Yaskawa INFORM job: DEMO_ROOF_UPPER_0625_3PAINT_3.JBI

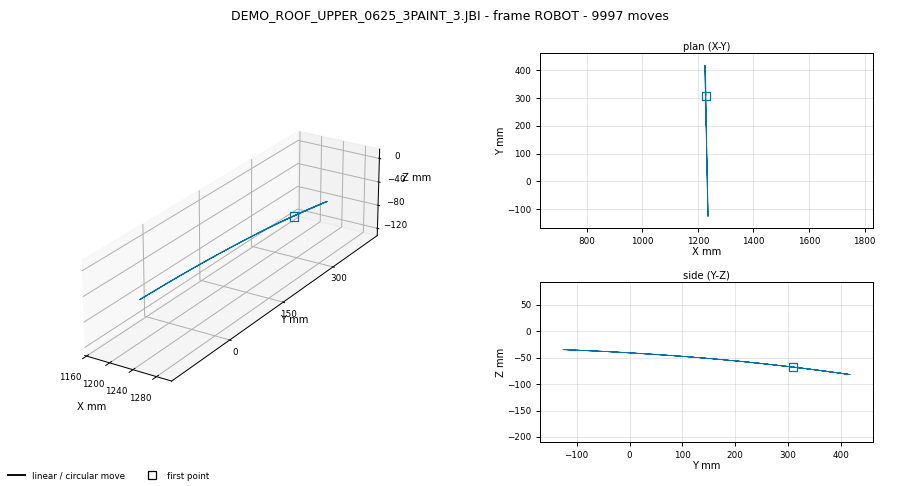
[picture p0: tool path of DEMO_ROOF_UPPER_0625_3PAINT_3.JBI in frame ROBOT, 9997 of 9997 moves have a stored position in this frame; points joined in program order, loops and branches not executed]
/JOB
//NAME DEMO_ROOF_UPPER_0625_3PAINT3
//POS
///NPOS 9997,0,0,0,0,0
///TOOL 0
///USER 0
///POSTYPE ROBOT
///RECTAN
///RCONF 1,0,0,0,0,0,0,0,0,0,0,0,0,0,0,0,0,0,0,0,0,0,0,0
C00000=1229.073,308.460,-67.633,-176.288,6.838,148.176
C00001=1229.069,308.709,-67.663,-176.286,6.841,148.176
C00002=1229.065,308.957,-67.692,-176.284,6.843,148.176
C00003=1229.061,309.205,-67.722,-176.281,6.846,148.176
C00004=1229.056,309.453,-67.752,-176.279,6.848,148.176
C00005=1229.052,309.701,-67.782,-176.277,6.850,148.176
C00006=1229.048,309.950,-67.811,-176.275,6.853,148.176
C00007=1229.044,310.198,-67.841,-176.272,6.856,148.176
C00008=1229.039,310.446,-67.871,-176.270,6.858,148.176
C00009=1229.035,310.694,-67.901,-176.268,6.860,148.176
C00010=1229.031,310.942,-67.930,-176.265,6.863,148.176
C00011=1229.026,311.190,-67.961,-176.263,6.865,148.176
C00012=1229.023,311.439,-67.991,-176.261,6.868,148.176
C00013=1229.019,311.687,-68.021,-176.258,6.871,148.176
C00014=1229.014,311.936,-68.051,-176.256,6.873,148.176
C00015=1229.010,312.184,-68.081,-176.254,6.875,148.176
C00016=1229.006,312.432,-68.111,-176.252,6.877,148.176
C00017=1229.001,312.680,-68.141,-176.249,6.880,148.176
C00018=1228.997,312.928,-68.171,-176.247,6.883,148.176
C00019=1228.992,313.176,-68.201,-176.245,6.885,148.176
C00020=1228.988,313.424,-68.231,-176.243,6.888,148.176
C00021=1228.984,313.672,-68.261,-176.241,6.890,148.176
C00022=1228.979,313.920,-68.291,-176.239,6.893,148.176
C00023=1228.975,314.168,-68.321,-176.237,6.895,148.176
C00024=1228.971,314.416,-68.352,-176.234,6.898,148.176
C00025=1228.966,314.665,-68.381,-176.232,6.900,148.176
C00026=1228.963,314.912,-68.411,-176.230,6.902,148.176
C00027=1228.957,315.189,-68.445,-176.227,6.905,148.176
C00028=1228.953,315.465,-68.478,-176.224,6.909,148.176
C00029=1228.948,315.741,-68.512,-176.222,6.911,148.176
C00030=1228.944,316.015,-68.545,-176.220,6.914,148.176
C00031=1228.939,316.264,-68.575,-176.218,6.916,148.176
C00032=1228.935,316.512,-68.606,-176.215,6.919,148.176
C00033=1228.931,316.761,-68.636,-176.213,6.922,148.176
C00034=1228.927,317.009,-68.666,-176.211,6.924,148.176
C00035=1228.922,317.257,-68.697,-176.209,6.927,148.176
C00036=1228.918,317.505,-68.726,-176.206,6.929,148.176
C00037=1228.913,317.753,-68.757,-176.204,6.931,148.176
C00038=1228.909,318.000,-68.787,-176.202,6.935,148.176
C00039=1228.905,318.250,-68.818,-176.200,6.937,148.176
C00040=1228.901,318.497,-68.848,-176.198,6.939,148.176
C00041=1228.897,318.745,-68.879,-176.196,6.941,148.176
C00042=1228.892,318.994,-68.908,-176.193,6.944,148.176
C00043=1228.888,319.242,-68.939,-176.192,6.947,148.176
C00044=1228.883,319.489,-68.970,-176.190,6.949,148.176
C00045=1228.880,319.738,-68.999,-176.187,6.952,148.176
C00046=1228.875,319.986,-69.030,-176.185,6.954,148.176
C00047=1228.871,320.234,-69.060,-176.183,6.957,148.176
C00048=1228.867,320.482,-69.091,-176.180,6.960,148.176
C00049=1228.863,320.730,-69.121,-176.178,6.962,148.176
C00050=1228.858,320.979,-69.152,-176.176,6.965,148.176
C00051=1228.854,321.227,-69.182,-176.174,6.968,148.176
C00052=1228.850,321.475,-69.213,-176.172,6.970,148.176
C00053=1228.845,321.722,-69.243,-176.170,6.972,148.176
C00054=1228.841,321.971,-69.275,-176.168,6.975,148.176
C00055=1228.837,322.219,-69.305,-176.165,6.978,148.176
C00056=1228.832,322.467,-69.335,-176.164,6.980,148.176
C00057=1228.829,322.715,-69.365,-176.161,6.982,148.176
C00058=1228.824,322.963,-69.396,-176.159,6.985,148.176
C00059=1228.820,323.212,-69.427,-176.157,6.988,148.176
C00060=1228.816,323.459,-69.457,-176.155,6.990,148.176
C00061=1228.811,323.707,-69.488,-176.152,6.993,148.176
C00062=1228.807,323.955,-69.519,-176.151,6.996,148.176
C00063=1228.803,324.204,-69.550,-176.149,6.998,148.176
C00064=1228.799,324.452,-69.580,-176.146,7.001,148.176
C00065=1228.794,324.699,-69.611,-176.144,7.003,148.176
C00066=1228.790,324.948,-69.642,-176.142,7.006,148.177
C00067=1228.786,325.196,-69.672,-176.140,7.008,148.177
C00068=1228.782,325.444,-69.703,-176.138,7.011,148.177
C00069=1228.777,325.692,-69.733,-176.136,7.014,148.177
C00070=1228.773,325.940,-69.765,-176.134,7.016,148.177
C00071=1228.769,326.188,-69.795,-176.132,7.019,148.177
C00072=1228.765,326.436,-69.825,-176.130,7.021,148.177
C00073=1228.761,326.685,-69.857,-176.127,7.024,148.177
C00074=1228.756,326.933,-69.887,-176.125,7.027,148.177
C00075=1228.752,327.180,-69.918,-176.123,7.029,148.177
C00076=1228.748,327.429,-69.949,-176.121,7.032,148.177
C00077=1228.744,327.677,-69.979,-176.119,7.035,148.177
C00078=1228.739,327.925,-70.010,-176.117,7.037,148.177
C00079=1228.735,328.173,-70.041,-176.115,7.040,148.177
C00080=1228.731,328.420,-70.072,-176.113,7.042,148.177
C00081=1228.727,328.668,-70.103,-176.111,7.045,148.177
C00082=1228.723,328.917,-70.134,-176.109,7.047,148.177
C00083=1228.718,329.165,-70.165,-176.107,7.050,148.177
C00084=1228.714,329.413,-70.196,-176.105,7.053,148.178
C00085=1228.710,329.662,-70.227,-176.102,7.055,148.178
C00086=1228.706,329.909,-70.258,-176.101,7.058,148.178
C00087=1228.701,330.157,-70.288,-176.098,7.061,148.178
C00088=1228.697,330.405,-70.320,-176.097,7.063,148.178
C00089=1228.693,330.653,-70.350,-176.094,7.066,148.178
C00090=1228.688,330.901,-70.382,-176.093,7.068,148.178
C00091=1228.684,331.149,-70.413,-176.090,7.071,148.178
C00092=1228.680,331.397,-70.444,-176.089,7.074,148.178
C00093=1228.676,331.646,-70.475,-176.086,7.076,148.178
C00094=1228.671,331.893,-70.506,-176.084,7.079,148.178
C00095=1228.667,332.141,-70.537,-176.082,7.082,148.178
C00096=1228.664,332.390,-70.568,-176.081,7.084,148.179
C00097=1228.659,332.637,-70.599,-176.078,7.087,148.179
C00098=1228.655,332.886,-70.630,-176.076,7.090,148.179
C00099=1228.651,333.133,-70.661,-176.074,7.092,148.179
C00100=1228.646,333.381,-70.692,-176.073,7.094,148.179
C00101=1228.642,333.629,-70.724,-176.070,7.098,148.179
C00102=1228.638,333.877,-70.754,-176.068,7.100,148.179
C00103=1228.634,334.125,-70.786,-176.066,7.102,148.179
C00104=1228.629,334.373,-70.817,-176.064,7.106,148.179
C00105=1228.625,334.622,-70.848,-176.062,7.108,148.179
C00106=1228.621,334.869,-70.880,-176.060,7.110,148.179
C00107=1228.616,335.117,-70.910,-176.058,7.114,148.180
C00108=1228.613,335.365,-70.942,-176.056,7.116,148.180
C00109=1228.608,335.613,-70.973,-176.054,7.119,148.180
C00110=1228.604,335.861,-71.005,-176.052,7.121,148.180
C00111=1228.600,336.109,-71.036,-176.050,7.124,148.180
C00112=1228.596,336.357,-71.067,-176.048,7.127,148.180
C00113=1228.591,336.605,-71.098,-176.046,7.129,148.180
C00114=1228.588,336.853,-71.130,-176.044,7.132,148.180
C00115=1228.583,337.101,-71.161,-176.042,7.134,148.180
C00116=1228.579,337.350,-71.193,-176.040,7.137,148.181
C00117=1228.574,337.598,-71.224,-176.039,7.140,148.181
C00118=1228.570,337.846,-71.256,-176.036,7.143,148.181
C00119=1228.566,338.094,-71.287,-176.035,7.145,148.181
C00120=1228.562,338.342,-71.318,-176.033,7.148,148.181
C00121=1228.557,338.590,-71.349,-176.030,7.151,148.181
C00122=1228.554,338.838,-71.381,-176.029,7.153,148.181
C00123=1228.549,339.085,-71.413,-176.027,7.156,148.181
C00124=1228.545,339.334,-71.444,-176.025,7.158,148.181
C00125=1228.541,339.581,-71.475,-176.023,7.161,148.182
C00126=1228.537,339.829,-71.508,-176.021,7.164,148.182
C00127=1228.532,340.077,-71.538,-176.020,7.166,148.182
C00128=1228.528,340.325,-71.570,-176.017,7.169,148.182
C00129=1228.524,340.573,-71.602,-176.015,7.172,148.182
C00130=1228.520,340.821,-71.633,-176.014,7.175,148.182
C00131=1228.516,341.099,-71.668,-176.011,7.178,148.182
C00132=1228.510,341.377,-71.704,-176.009,7.180,148.183
C00133=1228.505,341.654,-71.739,-176.007,7.184,148.183
C00134=1228.501,341.932,-71.775,-176.005,7.187,148.183
C00135=1228.497,342.180,-71.805,-176.003,7.189,148.183
C00136=1228.493,342.428,-71.837,-176.001,7.192,148.183
C00137=1228.488,342.675,-71.869,-175.999,7.195,148.183
C00138=1228.484,342.923,-71.901,-175.998,7.198,148.184
C00139=1228.480,343.171,-71.933,-175.996,7.200,148.184
C00140=1228.476,343.419,-71.964,-175.994,7.202,148.184
C00141=1228.471,343.668,-71.996,-175.992,7.206,148.184
C00142=1228.467,343.915,-72.028,-175.990,7.208,148.184
C00143=1228.463,344.163,-72.060,-175.988,7.211,148.184
C00144=1228.459,344.410,-72.091,-175.987,7.213,148.185
C00145=1228.454,344.659,-72.123,-175.984,7.216,148.185
C00146=1228.451,344.907,-72.155,-175.982,7.219,148.185
C00147=1228.446,345.155,-72.186,-175.981,7.221,148.185
C00148=1228.443,345.403,-72.218,-175.979,7.224,148.185
C00149=1228.437,345.651,-72.250,-175.977,7.227,148.185
C00150=1228.434,345.899,-72.282,-175.975,7.230,148.185
C00151=1228.430,346.147,-72.314,-175.974,7.232,148.186
C00152=1228.425,346.394,-72.346,-175.972,7.235,148.186
C00153=1228.421,346.643,-72.377,-175.970,7.238,148.186
C00154=1228.417,346.891,-72.409,-175.968,7.240,148.186
C00155=1228.412,347.139,-72.441,-175.966,7.243,148.186
C00156=1228.409,347.387,-72.473,-175.965,7.246,148.186
C00157=1228.404,347.634,-72.504,-175.962,7.249,148.187
C00158=1228.400,347.882,-72.537,-175.961,7.251,148.187
C00159=1228.396,348.130,-72.568,-175.959,7.254,148.187
C00160=1228.391,348.378,-72.601,-175.958,7.256,148.187
C00161=1228.387,348.626,-72.632,-175.955,7.260,148.187
C00162=1228.384,348.874,-72.664,-175.954,7.262,148.188
C00163=1228.379,349.122,-72.696,-175.952,7.265,148.188
C00164=1228.375,349.370,-72.728,-175.951,7.267,148.188
C00165=1228.370,349.618,-72.761,-175.949,7.270,148.188
C00166=1228.366,349.865,-72.792,-175.947,7.273,148.188
C00167=1228.362,350.113,-72.824,-175.945,7.276,148.189
C00168=1228.358,350.361,-72.857,-175.943,7.278,148.189
C00169=1228.355,350.609,-72.889,-175.942,7.281,148.189
C00170=1228.350,350.857,-72.921,-175.940,7.284,148.189
C00171=1228.346,351.105,-72.953,-175.938,7.287,148.189
C00172=1228.341,351.353,-72.985,-175.936,7.289,148.190
C00173=1228.337,351.601,-73.017,-175.935,7.292,148.190
C00174=1228.333,351.849,-73.049,-175.933,7.294,148.190
C00175=1228.329,352.097,-73.081,-175.931,7.298,148.190
C00176=1228.325,352.344,-73.113,-175.929,7.300,148.190
C00177=1228.320,352.592,-73.146,-175.928,7.303,148.190
C00178=1228.317,352.840,-73.178,-175.926,7.305,148.191
C00179=1228.312,353.088,-73.210,-175.924,7.308,148.191
C00180=1228.308,353.336,-73.241,-175.922,7.311,148.191
C00181=1228.304,353.584,-73.275,-175.921,7.314,148.191
C00182=1228.300,353.832,-73.306,-175.920,7.317,148.192
C00183=1228.296,354.080,-73.339,-175.918,7.319,148.192
C00184=1228.291,354.328,-73.371,-175.916,7.322,148.192
C00185=1228.287,354.576,-73.403,-175.914,7.325,148.192
C00186=1228.283,354.823,-73.436,-175.912,7.328,148.192
C00187=1228.279,355.071,-73.468,-175.911,7.330,148.193
C00188=1228.274,355.319,-73.500,-175.909,7.333,148.193
C00189=1228.271,355.566,-73.532,-175.908,7.335,148.193
C00190=1228.266,355.815,-73.565,-175.906,7.339,148.193
C00191=1228.263,356.063,-73.597,-175.904,7.341,148.194
C00192=1228.258,356.311,-73.630,-175.903,7.344,148.194
C00193=1228.253,356.558,-73.662,-175.901,7.346,148.194
C00194=1228.250,356.806,-73.694,-175.899,7.349,148.194
C00195=1228.246,357.054,-73.727,-175.898,7.352,148.195
C00196=1228.242,357.302,-73.759,-175.896,7.355,148.195
C00197=1228.237,357.550,-73.791,-175.894,7.358,148.195
C00198=1228.233,357.797,-73.824,-175.893,7.360,148.195
C00199=1228.229,358.045,-73.856,-175.892,7.363,148.196
C00200=1228.224,358.294,-73.888,-175.890,7.366,148.196
C00201=1228.220,358.542,-73.922,-175.888,7.368,148.196
C00202=1228.217,358.790,-73.953,-175.886,7.371,148.196
C00203=1228.212,359.037,-73.986,-175.885,7.374,148.197
C00204=1228.208,359.285,-74.018,-175.883,7.377,148.197
C00205=1228.204,359.532,-74.051,-175.882,7.379,148.197
C00206=1228.200,359.781,-74.084,-175.880,7.382,148.197
C00207=1228.196,360.028,-74.116,-175.879,7.385,148.198
C00208=1228.192,360.276,-74.149,-175.877,7.387,148.198
C00209=1228.187,360.523,-74.181,-175.875,7.391,148.198
C00210=1228.183,360.772,-74.213,-175.874,7.393,148.198
C00211=1228.179,361.019,-74.246,-175.872,7.396,148.199
C00212=1228.175,361.268,-74.279,-175.871,7.398,148.199
C00213=1228.171,361.515,-74.312,-175.870,7.401,148.199
C00214=1228.167,361.763,-74.344,-175.868,7.404,148.199
C00215=1228.163,362.011,-74.377,-175.866,7.406,148.200
C00216=1228.158,362.259,-74.409,-175.865,7.409,148.200
C00217=1228.154,362.506,-74.442,-175.863,7.413,148.200
C00218=1228.150,362.755,-74.474,-175.862,7.415,148.201
C00219=1228.146,363.002,-74.507,-175.860,7.418,148.201
C00220=1228.142,363.250,-74.540,-175.859,7.420,148.201
C00221=1228.138,363.498,-74.572,-175.857,7.423,148.201
C00222=1228.134,363.746,-74.605,-175.856,7.426,148.202
C00223=1228.129,363.994,-74.638,-175.855,7.429,148.202
C00224=1228.125,364.242,-74.671,-175.853,7.431,148.202
C00225=1228.121,364.490,-74.704,-175.852,7.434,148.202
C00226=1228.117,364.737,-74.736,-175.850,7.436,148.203
C00227=1228.113,364.985,-74.769,-175.848,7.440,148.203
C00228=1228.108,365.232,-74.802,-175.847,7.443,148.203
C00229=1228.104,365.481,-74.834,-175.845,7.445,148.204
C00230=1228.100,365.728,-74.867,-175.844,7.448,148.204
C00231=1228.096,365.976,-74.900,-175.842,7.451,148.204
C00232=1228.092,366.224,-74.933,-175.841,7.453,148.204
C00233=1228.088,366.472,-74.966,-175.840,7.456,148.205
C00234=1228.084,366.720,-74.999,-175.838,7.459,148.205
C00235=1228.079,366.999,-75.036,-175.837,7.461,148.205
C00236=1228.074,367.278,-75.072,-175.835,7.465,148.206
C00237=1228.070,367.558,-75.110,-175.834,7.468,148.206
C00238=1228.065,367.838,-75.147,-175.832,7.471,148.206
C00239=1228.061,368.086,-75.180,-175.831,7.474,148.207
C00240=1228.057,368.334,-75.213,-175.829,7.476,148.207
C00241=1228.052,368.581,-75.246,-175.828,7.479,148.207
C00242=1228.049,368.829,-75.279,-175.827,7.482,148.208
C00243=1228.045,369.077,-75.312,-175.825,7.485,148.208
C00244=1228.040,369.325,-75.344,-175.824,7.487,148.208
C00245=1228.036,369.573,-75.377,-175.822,7.490,148.209
C00246=1228.032,369.820,-75.410,-175.821,7.493,148.209
C00247=1228.028,370.068,-75.444,-175.820,7.496,148.209
C00248=1228.024,370.316,-75.477,-175.818,7.498,148.210
C00249=1228.020,370.564,-75.510,-175.817,7.501,148.210
C00250=1228.016,370.811,-75.543,-175.816,7.504,148.210
C00251=1228.011,371.059,-75.576,-175.814,7.506,148.210
C00252=1228.007,371.307,-75.609,-175.813,7.509,148.211
C00253=1228.003,371.555,-75.642,-175.812,7.512,148.211
C00254=1227.999,371.803,-75.675,-175.810,7.515,148.211
C00255=1227.995,372.051,-75.708,-175.809,7.517,148.212
C00256=1227.990,372.298,-75.741,-175.809,7.519,148.212
C00257=1227.986,372.546,-75.774,-175.807,7.522,148.212
C00258=1227.982,372.794,-75.808,-175.806,7.525,148.213
C00259=1227.979,373.041,-75.840,-175.805,7.528,148.213
C00260=1227.975,373.289,-75.873,-175.803,7.530,148.214
C00261=1227.971,373.537,-75.907,-175.802,7.533,148.214
C00262=1227.966,373.784,-75.940,-175.801,7.536,148.214
C00263=1227.962,374.032,-75.973,-175.800,7.539,148.215
C00264=1227.958,374.280,-76.006,-175.798,7.541,148.215
C00265=1227.953,374.528,-76.040,-175.797,7.544,148.215
C00266=1227.949,374.776,-76.073,-175.796,7.547,148.216
C00267=1227.945,375.023,-76.106,-175.794,7.550,148.216
C00268=1227.941,375.271,-76.139,-175.793,7.552,148.216
C00269=1227.937,375.519,-76.172,-175.793,7.554,148.217
C00270=1227.933,375.766,-76.205,-175.791,7.557,148.217
C00271=1227.928,376.014,-76.239,-175.790,7.560,148.217
C00272=1227.924,376.262,-76.272,-175.789,7.563,148.218
C00273=1227.920,376.510,-76.305,-175.787,7.565,148.218
C00274=1227.916,376.757,-76.338,-175.786,7.568,148.218
C00275=1227.913,377.005,-76.372,-175.785,7.571,148.219
C00276=1227.909,377.253,-76.406,-175.783,7.574,148.219
C00277=1227.905,377.501,-76.439,-175.783,7.575,148.219
C00278=1227.900,377.748,-76.472,-175.782,7.578,148.220
C00279=1227.896,377.996,-76.505,-175.781,7.581,148.220
C00280=1227.892,378.244,-76.538,-175.779,7.584,148.221
C00281=1227.887,378.492,-76.572,-175.778,7.587,148.221
C00282=1227.883,378.740,-76.605,-175.777,7.590,148.221
C00283=1227.879,378.987,-76.639,-175.776,7.592,148.222
C00284=1227.875,379.234,-76.672,-175.775,7.594,148.222
C00285=1227.871,379.482,-76.705,-175.774,7.597,148.222
C00286=1227.867,379.731,-76.739,-175.772,7.600,148.223
C00287=1227.863,379.978,-76.772,-175.771,7.603,148.223
C00288=1227.859,380.225,-76.806,-175.771,7.605,148.223
C00289=1227.855,380.474,-76.840,-175.769,7.607,148.224
C00290=1227.850,380.721,-76.873,-175.768,7.610,148.224
C00291=1227.846,380.969,-76.906,-175.767,7.613,148.225
C00292=1227.842,381.217,-76.939,-175.767,7.615,148.225
C00293=1227.838,381.464,-76.973,-175.765,7.618,148.225
C00294=1227.834,381.712,-77.006,-175.764,7.621,148.226
C00295=1227.830,381.960,-77.040,-175.763,7.623,148.226
C00296=1227.826,382.207,-77.074,-175.762,7.626,148.227
C00297=1227.822,382.455,-77.107,-175.761,7.628,148.227
C00298=1227.818,382.703,-77.140,-175.760,7.631,148.227
C00299=1227.814,382.951,-77.173,-175.759,7.634,148.228
C00300=1227.809,383.198,-77.208,-175.758,7.636,148.228
C00301=1227.805,383.446,-77.241,-175.757,7.639,148.228
C00302=1227.801,383.694,-77.275,-175.756,7.642,148.229
C00303=1227.798,383.941,-77.308,-175.755,7.644,148.229
C00304=1227.793,384.189,-77.342,-175.754,7.646,148.230
C00305=1227.789,384.437,-77.375,-175.753,7.649,148.230
C00306=1227.785,384.684,-77.409,-175.752,7.652,148.230
C00307=1227.781,384.932,-77.442,-175.751,7.654,148.231
C00308=1227.777,385.180,-77.476,-175.750,7.657,148.231
C00309=1227.773,385.428,-77.510,-175.749,7.660,148.232
C00310=1227.768,385.675,-77.544,-175.748,7.662,148.232
C00311=1227.765,385.923,-77.577,-175.747,7.664,148.232
C00312=1227.760,386.170,-77.611,-175.746,7.667,148.233
C00313=1227.756,386.418,-77.644,-175.745,7.670,148.233
C00314=1227.752,386.666,-77.679,-175.744,7.672,148.233
C00315=1227.748,386.914,-77.712,-175.743,7.675,148.234
C00316=1227.744,387.161,-77.746,-175.743,7.677,148.234
C00317=1227.739,387.409,-77.779,-175.742,7.680,148.235
C00318=1227.735,387.657,-77.813,-175.740,7.683,148.235
C00319=1227.732,387.905,-77.847,-175.740,7.685,148.236
C00320=1227.727,388.153,-77.881,-175.739,7.688,148.236
C00321=1227.723,388.400,-77.914,-175.737,7.690,148.236
C00322=1227.719,388.647,-77.948,-175.737,7.692,148.237
C00323=1227.715,388.895,-77.982,-175.736,7.695,148.237
C00324=1227.711,389.143,-78.016,-175.734,7.698,148.237
C00325=1227.707,389.390,-78.049,-175.734,7.700,148.238
C00326=1227.702,389.638,-78.083,-175.733,7.703,148.238
C00327=1227.699,389.886,-78.117,-175.732,7.705,148.239
C00328=1227.694,390.133,-78.150,-175.731,7.708,148.239
C00329=1227.690,390.381,-78.185,-175.731,7.710,148.240
C00330=1227.686,390.629,-78.218,-175.729,7.713,148.240
C00331=1227.683,390.876,-78.252,-175.728,7.716,148.240
C00332=1227.678,391.124,-78.286,-175.728,7.718,148.241
C00333=1227.674,391.372,-78.320,-175.727,7.721,148.241
C00334=1227.671,391.619,-78.354,-175.726,7.723,148.242
C00335=1227.666,391.867,-78.388,-175.725,7.726,148.242
C00336=1227.662,392.114,-78.422,-175.725,7.727,148.242
C00337=1227.658,392.363,-78.456,-175.723,7.730,148.243
C00338=1227.654,392.610,-78.490,-175.723,7.733,148.243
C00339=1227.649,392.892,-78.528,-175.722,7.735,148.244
C00340=1227.645,393.173,-78.566,-175.721,7.738,148.244
C00341=1227.640,393.454,-78.606,-175.720,7.741,148.245
C00342=1227.635,393.736,-78.644,-175.719,7.744,148.245
C00343=1227.631,393.983,-78.678,-175.718,7.746,148.245
C00344=1227.627,394.231,-78.711,-175.717,7.749,148.246
C00345=1227.623,394.479,-78.745,-175.717,7.751,148.246
C00346=1227.619,394.726,-78.779,-175.716,7.754,148.247
C00347=1227.615,394.974,-78.813,-175.715,7.756,148.247
C00348=1227.611,395.222,-78.847,-175.714,7.759,148.248
C00349=1227.607,395.470,-78.882,-175.714,7.761,148.248
C00350=1227.603,395.717,-78.915,-175.713,7.764,148.248
C00351=1227.598,395.965,-78.950,-175.712,7.766,148.249
C00352=1227.594,396.212,-78.983,-175.711,7.769,148.249
C00353=1227.590,396.461,-79.018,-175.710,7.771,148.250
C00354=1227.586,396.708,-79.051,-175.710,7.774,148.250
C00355=1227.582,396.955,-79.085,-175.709,7.776,148.251
C00356=1227.578,397.203,-79.120,-175.708,7.779,148.251
C00357=1227.574,397.451,-79.153,-175.707,7.781,148.251
C00358=1227.570,397.698,-79.188,-175.707,7.783,148.252
C00359=1227.566,397.945,-79.222,-175.706,7.786,148.252
C00360=1227.562,398.193,-79.256,-175.705,7.788,148.253
C00361=1227.558,398.441,-79.290,-175.704,7.791,148.253
C00362=1227.553,398.689,-79.324,-175.704,7.793,148.253
C00363=1227.550,398.936,-79.358,-175.703,7.795,148.254
C00364=1227.545,399.184,-79.393,-175.702,7.798,148.254
C00365=1227.541,399.431,-79.426,-175.701,7.800,148.255
C00366=1227.537,399.680,-79.461,-175.701,7.803,148.255
C00367=1227.533,399.927,-79.495,-175.700,7.805,148.256
C00368=1227.529,400.174,-79.529,-175.699,7.807,148.256
C00369=1227.526,400.422,-79.563,-175.699,7.810,148.256
C00370=1227.521,400.670,-79.597,-175.698,7.812,148.257
C00371=1227.517,400.917,-79.631,-175.697,7.815,148.257
C00372=1227.513,401.165,-79.666,-175.696,7.817,148.258
C00373=1227.508,401.413,-79.700,-175.696,7.819,148.258
C00374=1227.505,401.660,-79.734,-175.695,7.822,148.258
C00375=1227.501,401.908,-79.769,-175.694,7.824,148.259
C00376=1227.496,402.156,-79.802,-175.694,7.826,148.259
C00377=1227.492,402.403,-79.837,-175.693,7.829,148.260
C00378=1227.489,402.651,-79.871,-175.692,7.831,148.260
C00379=1227.484,402.898,-79.905,-175.692,7.833,148.260
C00380=1227.480,403.145,-79.939,-175.691,7.836,148.261
C00381=1227.476,403.393,-79.974,-175.690,7.838,148.261
C00382=1227.472,403.641,-80.008,-175.690,7.840,148.262
C00383=1227.468,403.889,-80.043,-175.689,7.842,148.262
C00384=1227.464,404.137,-80.076,-175.688,7.845,148.263
C00385=1227.460,404.384,-80.110,-175.688,7.847,148.263
C00386=1227.456,404.632,-80.145,-175.687,7.849,148.263
C00387=1227.451,404.879,-80.180,-175.686,7.852,148.264
C00388=1227.447,405.126,-80.213,-175.686,7.854,148.264
C00389=1227.443,405.375,-80.248,-175.685,7.856,148.265
C00390=1227.440,405.622,-80.282,-175.685,7.858,148.265
C00391=1227.435,405.869,-80.317,-175.684,7.861,148.266
C00392=1227.431,406.117,-80.351,-175.683,7.863,148.266
C00393=1227.427,406.364,-80.385,-175.682,7.865,148.266
C00394=1227.423,406.613,-80.420,-175.682,7.868,148.267
C00395=1227.419,406.860,-80.454,-175.681,7.870,148.267
C00396=1227.415,407.107,-80.489,-175.680,7.872,148.268
C00397=1227.411,407.355,-80.523,-175.680,7.874,148.268
C00398=1227.407,407.602,-80.557,-175.679,7.877,148.269
C00399=1227.403,407.850,-80.592,-175.678,7.879,148.269
C00400=1227.398,408.098,-80.627,-175.678,7.881,148.269
C00401=1227.395,408.345,-80.660,-175.678,7.883,148.270
C00402=1227.391,408.593,-80.695,-175.677,7.885,148.270
C00403=1227.386,408.840,-80.730,-175.676,7.888,148.271
C00404=1227.383,409.088,-80.764,-175.676,7.890,148.271
C00405=1227.378,409.336,-80.798,-175.675,7.892,148.271
C00406=1227.375,409.583,-80.833,-175.674,7.894,148.272
C00407=1227.371,409.831,-80.867,-175.674,7.897,148.272
C00408=1227.366,410.078,-80.902,-175.673,7.899,148.273
C00409=1227.363,410.326,-80.936,-175.672,7.901,148.273
C00410=1227.358,410.574,-80.970,-175.672,7.904,148.274
C00411=1227.354,410.822,-81.005,-175.672,7.906,148.274
C00412=1227.350,411.069,-81.040,-175.671,7.908,148.274
C00413=1227.346,411.317,-81.074,-175.670,7.911,148.275
C00414=1227.342,411.564,-81.108,-175.670,7.913,148.275
C00415=1227.337,411.812,-81.143,-175.669,7.915,148.275
C00416=1227.334,412.059,-81.178,-175.668,7.917,148.276
C00417=1227.330,412.306,-81.212,-175.668,7.919,148.276
C00418=1227.326,412.554,-81.247,-175.667,7.921,148.277
C00419=1227.322,412.802,-81.281,-175.666,7.924,148.277
C00420=1227.318,413.050,-81.316,-175.666,7.926,148.278
C00421=1227.313,413.297,-81.350,-175.665,7.928,148.278
C00422=1227.309,413.545,-81.385,-175.665,7.930,148.278
C00423=1227.306,413.792,-81.419,-175.665,7.932,148.279
C00424=1227.301,414.039,-81.454,-175.664,7.934,148.279
C00425=1227.297,414.287,-81.489,-175.663,7.936,148.280
C00426=1227.293,414.535,-81.523,-175.662,7.939,148.280
C00427=1227.290,414.783,-81.558,-175.662,7.941,148.281
C00428=1227.285,415.030,-81.592,-175.661,7.943,148.281
C00429=1227.281,415.278,-81.627,-175.661,7.945,148.281
C00430=1227.277,415.525,-81.662,-175.661,7.948,148.282
C00431=1227.270,415.917,-81.717,-175.660,7.951,148.282
C00432=1227.264,416.309,-81.771,-175.659,7.955,148.283
C00433=1227.258,416.701,-81.826,-175.658,7.958,148.284
C00434=1227.253,417.094,-81.881,-175.657,7.961,148.284
C00435=1226.832,417.093,-81.914,-175.660,7.971,148.288
C00436=1226.835,416.698,-81.859,-175.661,7.968,148.287
C00437=1226.843,416.304,-81.804,-175.662,7.965,148.287
C00438=1226.849,415.909,-81.748,-175.663,7.961,148.286
C00439=1226.855,415.514,-81.693,-175.664,7.958,148.285
C00440=1226.859,415.267,-81.659,-175.664,7.956,148.285
C00441=1226.863,415.020,-81.625,-175.665,7.954,148.285
C00442=1226.867,414.772,-81.589,-175.665,7.952,148.284
C00443=1226.871,414.525,-81.555,-175.666,7.949,148.284
C00444=1226.875,414.277,-81.520,-175.667,7.947,148.283
C00445=1226.879,414.030,-81.486,-175.667,7.945,148.283
C00446=1226.883,413.781,-81.451,-175.668,7.943,148.282
C00447=1226.888,413.534,-81.417,-175.668,7.941,148.282
C00448=1226.892,413.286,-81.382,-175.669,7.938,148.282
C00449=1226.895,413.039,-81.347,-175.669,7.936,148.281
C00450=1226.899,412.791,-81.312,-175.670,7.934,148.281
C00451=1226.904,412.544,-81.278,-175.671,7.931,148.280
C00452=1226.908,412.296,-81.243,-175.671,7.929,148.280
C00453=1226.912,412.049,-81.209,-175.672,7.927,148.280
C00454=1226.916,411.801,-81.175,-175.672,7.925,148.279
C00455=1226.920,411.553,-81.140,-175.673,7.923,148.279
C00456=1226.924,411.306,-81.106,-175.674,7.920,148.278
C00457=1226.928,411.058,-81.071,-175.674,7.918,148.278
C00458=1226.932,410.811,-81.036,-175.675,7.916,148.277
C00459=1226.935,410.563,-81.002,-175.675,7.914,148.277
C00460=1226.940,410.316,-80.967,-175.676,7.912,148.277
C00461=1226.945,410.068,-80.933,-175.676,7.910,148.276
C00462=1226.949,409.820,-80.898,-175.677,7.907,148.276
C00463=1226.952,409.573,-80.864,-175.678,7.905,148.275
C00464=1226.956,409.325,-80.829,-175.678,7.903,148.275
C00465=1226.961,409.078,-80.795,-175.679,7.901,148.275
C00466=1226.964,408.830,-80.761,-175.679,7.899,148.274
C00467=1226.969,408.582,-80.726,-175.680,7.896,148.274
C00468=1226.973,408.335,-80.692,-175.681,7.894,148.273
C00469=1226.977,408.087,-80.657,-175.681,7.892,148.273
C00470=1226.981,407.840,-80.623,-175.682,7.890,148.273
C00471=1226.984,407.592,-80.589,-175.683,7.887,148.272
C00472=1226.989,407.345,-80.554,-175.683,7.885,148.272
C00473=1226.993,407.097,-80.520,-175.684,7.883,148.271
C00474=1226.997,406.849,-80.486,-175.684,7.880,148.271
C00475=1227.001,406.602,-80.451,-175.685,7.878,148.270
C00476=1227.005,406.354,-80.416,-175.686,7.876,148.270
C00477=1227.009,406.107,-80.382,-175.686,7.873,148.270
C00478=1227.014,405.859,-80.348,-175.687,7.871,148.269
C00479=1227.017,405.611,-80.314,-175.688,7.868,148.269
C00480=1227.021,405.364,-80.279,-175.688,7.866,148.268
C00481=1227.026,405.117,-80.245,-175.689,7.864,148.268
C00482=1227.029,404.869,-80.211,-175.689,7.862,148.268
C00483=1227.034,404.621,-80.176,-175.691,7.859,148.267
C00484=1227.037,404.374,-80.142,-175.691,7.857,148.267
C00485=1227.042,404.126,-80.107,-175.691,7.855,148.266
C00486=1227.046,403.878,-80.074,-175.693,7.852,148.266
C00487=1227.050,403.630,-80.039,-175.693,7.850,148.265
C00488=1227.054,403.383,-80.005,-175.693,7.848,148.265
C00489=1227.058,403.136,-79.971,-175.694,7.846,148.265
C00490=1227.062,402.888,-79.936,-175.695,7.843,148.264
C00491=1227.067,402.640,-79.902,-175.695,7.841,148.264
C00492=1227.070,402.392,-79.868,-175.696,7.839,148.263
C00493=1227.074,402.145,-79.833,-175.697,7.836,148.263
C00494=1227.078,401.898,-79.799,-175.697,7.834,148.262
C00495=1227.083,401.649,-79.765,-175.698,7.832,148.262
C00496=1227.086,401.402,-79.731,-175.699,7.829,148.262
C00497=1227.091,401.155,-79.697,-175.699,7.827,148.261
C00498=1227.094,400.907,-79.663,-175.700,7.824,148.261
C00499=1227.099,400.659,-79.628,-175.701,7.822,148.260
C00500=1227.103,400.412,-79.594,-175.702,7.820,148.260
C00501=1227.107,400.164,-79.560,-175.702,7.817,148.259
C00502=1227.111,399.916,-79.526,-175.703,7.815,148.259
C00503=1227.115,399.669,-79.492,-175.704,7.813,148.259
C00504=1227.119,399.421,-79.457,-175.704,7.810,148.258
C00505=1227.123,399.174,-79.423,-175.705,7.808,148.258
C00506=1227.128,398.926,-79.389,-175.706,7.805,148.257
C00507=1227.131,398.678,-79.355,-175.707,7.803,148.257
C00508=1227.136,398.431,-79.321,-175.707,7.801,148.257
C00509=1227.140,398.183,-79.287,-175.708,7.798,148.256
C00510=1227.144,397.935,-79.253,-175.709,7.796,148.256
C00511=1227.148,397.688,-79.219,-175.710,7.793,148.255
C00512=1227.152,397.440,-79.184,-175.710,7.791,148.255
C00513=1227.156,397.193,-79.150,-175.711,7.789,148.255
C00514=1227.160,396.944,-79.116,-175.712,7.786,148.254
C00515=1227.164,396.697,-79.082,-175.713,7.784,148.254
C00516=1227.168,396.450,-79.049,-175.713,7.781,148.253
C00517=1227.172,396.202,-79.014,-175.714,7.779,148.253
C00518=1227.176,395.954,-78.981,-175.715,7.776,148.252
C00519=1227.181,395.707,-78.946,-175.716,7.774,148.252
C00520=1227.185,395.460,-78.912,-175.716,7.771,148.251
C00521=1227.189,395.211,-78.878,-175.717,7.769,148.251
C00522=1227.193,394.964,-78.844,-175.718,7.766,148.251
C00523=1227.197,394.716,-78.810,-175.719,7.764,148.250
C00524=1227.201,394.468,-78.776,-175.720,7.761,148.250
C00525=1227.205,394.221,-78.742,-175.720,7.759,148.249
C00526=1227.209,393.973,-78.708,-175.721,7.756,148.249
C00527=1227.213,393.726,-78.675,-175.722,7.755,148.249
C00528=1227.217,393.444,-78.636,-175.723,7.751,148.248
C00529=1227.223,393.162,-78.597,-175.724,7.749,148.248
C00530=1227.227,392.882,-78.559,-175.725,7.746,148.247
C00531=1227.232,392.600,-78.520,-175.726,7.743,148.247
C00532=1227.236,392.352,-78.486,-175.726,7.741,148.246
C00533=1227.240,392.104,-78.452,-175.728,7.738,148.246
C00534=1227.244,391.857,-78.419,-175.728,7.736,148.246
C00535=1227.248,391.609,-78.384,-175.729,7.733,148.245
C00536=1227.252,391.361,-78.351,-175.730,7.731,148.245
C00537=1227.256,391.114,-78.317,-175.731,7.728,148.244
C00538=1227.260,390.866,-78.282,-175.731,7.726,148.244
C00539=1227.264,390.619,-78.249,-175.733,7.723,148.244
C00540=1227.269,390.371,-78.215,-175.734,7.720,148.243
C00541=1227.272,390.123,-78.181,-175.734,7.718,148.243
C00542=1227.276,389.876,-78.147,-175.735,7.715,148.242
C00543=1227.281,389.628,-78.114,-175.736,7.713,148.242
C00544=1227.285,389.380,-78.080,-175.737,7.710,148.241
C00545=1227.289,389.132,-78.046,-175.738,7.708,148.241
C00546=1227.293,388.885,-78.012,-175.739,7.706,148.241
C00547=1227.297,388.637,-77.979,-175.740,7.703,148.240
C00548=1227.301,388.390,-77.945,-175.741,7.701,148.240
C00549=1227.305,388.142,-77.911,-175.742,7.698,148.240
C00550=1227.309,387.894,-77.877,-175.742,7.695,148.239
C00551=1227.313,387.646,-77.843,-175.743,7.693,148.239
C00552=1227.317,387.399,-77.810,-175.744,7.690,148.238
C00553=1227.322,387.151,-77.776,-175.745,7.687,148.238
C00554=1227.326,386.903,-77.743,-175.746,7.685,148.237
C00555=1227.329,386.655,-77.708,-175.747,7.682,148.237
C00556=1227.334,386.407,-77.675,-175.748,7.680,148.237
C00557=1227.338,386.160,-77.641,-175.749,7.678,148.236
C00558=1227.342,385.913,-77.608,-175.750,7.675,148.236
C00559=1227.346,385.665,-77.574,-175.751,7.672,148.236
C00560=1227.350,385.417,-77.540,-175.752,7.670,148.235
C00561=1227.355,385.169,-77.507,-175.753,7.667,148.235
C00562=1227.358,384.922,-77.473,-175.754,7.664,148.234
C00563=1227.362,384.674,-77.440,-175.754,7.662,148.234
C00564=1227.367,384.426,-77.406,-175.756,7.659,148.233
C00565=1227.371,384.179,-77.372,-175.757,7.656,148.233
C00566=1227.375,383.931,-77.338,-175.758,7.654,148.233
C00567=1227.379,383.683,-77.305,-175.759,7.652,148.232
C00568=1227.383,383.435,-77.271,-175.760,7.649,148.232
C00569=1227.388,383.188,-77.238,-175.761,7.646,148.232
C00570=1227.392,382.940,-77.204,-175.762,7.644,148.231
C00571=1227.396,382.693,-77.171,-175.763,7.641,148.231
C00572=1227.400,382.445,-77.137,-175.764,7.638,148.230
C00573=1227.404,382.196,-77.103,-175.765,7.636,148.230
C00574=1227.408,381.949,-77.069,-175.766,7.634,148.230
C00575=1227.412,381.702,-77.036,-175.767,7.631,148.229
C00576=1227.416,381.454,-77.003,-175.768,7.628,148.229
C00577=1227.420,381.206,-76.970,-175.769,7.625,148.228
C00578=1227.424,380.959,-76.936,-175.770,7.623,148.228
C00579=1227.429,380.711,-76.902,-175.771,7.620,148.228
C00580=1227.433,380.463,-76.869,-175.772,7.617,148.227
C00581=1227.437,380.215,-76.836,-175.773,7.615,148.227
C00582=1227.440,379.968,-76.802,-175.775,7.612,148.227
C00583=1227.445,379.720,-76.769,-175.776,7.610,148.226
C00584=1227.449,379.472,-76.735,-175.777,7.607,148.226
C00585=1227.454,379.224,-76.702,-175.778,7.604,148.226
C00586=1227.458,378.976,-76.669,-175.779,7.602,148.225
C00587=1227.462,378.729,-76.635,-175.780,7.599,148.225
C00588=1227.466,378.482,-76.602,-175.781,7.596,148.224
C00589=1227.470,378.234,-76.568,-175.782,7.594,148.224
C00590=1227.474,377.986,-76.535,-175.783,7.591,148.224
C00591=1227.477,377.738,-76.502,-175.784,7.588,148.223
C00592=1227.482,377.490,-76.469,-175.786,7.586,148.223
C00593=1227.486,377.242,-76.435,-175.787,7.583,148.223
C00594=1227.491,376.994,-76.402,-175.788,7.580,148.222
C00595=1227.494,376.747,-76.368,-175.789,7.578,148.222
C00596=1227.499,376.499,-76.335,-175.790,7.575,148.222
C00597=1227.503,376.252,-76.301,-175.791,7.573,148.221
C00598=1227.507,376.004,-76.268,-175.792,7.570,148.221
C00599=1227.511,375.756,-76.235,-175.794,7.567,148.221
C00600=1227.515,375.508,-76.202,-175.795,7.564,148.220
C00601=1227.519,375.261,-76.169,-175.796,7.562,148.220
C00602=1227.523,375.013,-76.136,-175.798,7.559,148.219
C00603=1227.528,374.765,-76.103,-175.799,7.556,148.219
C00604=1227.532,374.518,-76.069,-175.800,7.554,148.219
C00605=1227.536,374.270,-76.036,-175.801,7.551,148.218
C00606=1227.540,374.022,-76.003,-175.802,7.549,148.218
C00607=1227.544,373.774,-75.970,-175.803,7.546,148.218
C00608=1227.548,373.526,-75.936,-175.805,7.543,148.217
C00609=1227.552,373.278,-75.903,-175.806,7.540,148.217
C00610=1227.556,373.030,-75.870,-175.807,7.538,148.217
C00611=1227.560,372.783,-75.837,-175.809,7.535,148.216
C00612=1227.564,372.535,-75.804,-175.810,7.532,148.216
C00613=1227.568,372.287,-75.771,-175.811,7.529,148.216
C00614=1227.572,372.040,-75.737,-175.812,7.527,148.215
C00615=1227.577,371.792,-75.704,-175.814,7.524,148.215
C00616=1227.581,371.544,-75.671,-175.815,7.521,148.215
C00617=1227.585,371.296,-75.638,-175.816,7.518,148.214
C00618=1227.589,371.049,-75.605,-175.818,7.516,148.214
C00619=1227.593,370.801,-75.572,-175.819,7.513,148.214
C00620=1227.597,370.553,-75.539,-175.820,7.510,148.213
C00621=1227.602,370.305,-75.506,-175.822,7.507,148.213
C00622=1227.606,370.057,-75.473,-175.823,7.505,148.213
C00623=1227.610,369.809,-75.440,-175.824,7.502,148.212
C00624=1227.613,369.562,-75.407,-175.826,7.499,148.212
C00625=1227.618,369.314,-75.374,-175.827,7.497,148.212
C00626=1227.622,369.066,-75.341,-175.828,7.494,148.211
C00627=1227.626,368.819,-75.308,-175.830,7.491,148.211
C00628=1227.630,368.570,-75.275,-175.831,7.489,148.211
C00629=1227.635,368.323,-75.243,-175.832,7.486,148.210
C00630=1227.639,368.076,-75.209,-175.834,7.483,148.210
C00631=1227.643,367.828,-75.176,-175.835,7.480,148.210
C00632=1227.648,367.548,-75.139,-175.837,7.478,148.210
C00633=1227.652,367.268,-75.102,-175.838,7.474,148.209
C00634=1227.657,366.989,-75.065,-175.840,7.471,148.209
C00635=1227.662,366.709,-75.028,-175.841,7.469,148.208
C00636=1227.666,366.461,-74.995,-175.843,7.465,148.208
C00637=1227.670,366.213,-74.962,-175.845,7.463,148.208
C00638=1227.673,365.966,-74.929,-175.846,7.460,148.207
C00639=1227.678,365.718,-74.897,-175.847,7.457,148.207
C00640=1227.682,365.470,-74.864,-175.849,7.454,148.207
C00641=1227.687,365.223,-74.831,-175.850,7.452,148.207
C00642=1227.691,364.974,-74.798,-175.851,7.449,148.206
C00643=1227.694,364.727,-74.766,-175.853,7.447,148.206
C00644=1227.699,364.479,-74.733,-175.854,7.444,148.206
C00645=1227.703,364.231,-74.700,-175.856,7.441,148.206
C00646=1227.707,363.983,-74.667,-175.857,7.439,148.205
C00647=1227.711,363.735,-74.634,-175.859,7.436,148.205
C00648=1227.715,363.487,-74.602,-175.861,7.432,148.205
C00649=1227.719,363.240,-74.569,-175.862,7.430,148.204
C00650=1227.724,362.993,-74.536,-175.863,7.427,148.204
C00651=1227.728,362.744,-74.504,-175.865,7.424,148.204
C00652=1227.732,362.497,-74.471,-175.866,7.422,148.204
C00653=1227.736,362.248,-74.439,-175.868,7.419,148.203
C00654=1227.740,362.001,-74.406,-175.869,7.416,148.203
C00655=1227.745,361.752,-74.373,-175.871,7.414,148.203
C00656=1227.748,361.505,-74.341,-175.872,7.411,148.203
C00657=1227.752,361.257,-74.307,-175.874,7.408,148.202
C00658=1227.757,361.010,-74.275,-175.876,7.405,148.202
C00659=1227.761,360.762,-74.243,-175.877,7.402,148.202
C00660=1227.765,360.514,-74.210,-175.878,7.400,148.201
C00661=1227.769,360.266,-74.177,-175.880,7.397,148.201
C00662=1227.773,360.018,-74.145,-175.882,7.395,148.201
C00663=1227.777,359.770,-74.112,-175.883,7.392,148.201
C00664=1227.782,359.522,-74.080,-175.885,7.389,148.200
C00665=1227.786,359.275,-74.048,-175.887,7.386,148.200
C00666=1227.790,359.027,-74.015,-175.888,7.383,148.200
C00667=1227.794,358.779,-73.983,-175.889,7.381,148.200
C00668=1227.798,358.531,-73.950,-175.891,7.378,148.199
C00669=1227.802,358.283,-73.918,-175.893,7.376,148.199
C00670=1227.806,358.035,-73.884,-175.894,7.372,148.199
C00671=1227.811,357.788,-73.853,-175.896,7.369,148.199
C00672=1227.815,357.539,-73.821,-175.898,7.367,148.198
C00673=1227.819,357.292,-73.787,-175.899,7.364,148.198
C00674=1227.823,357.044,-73.756,-175.900,7.362,148.198
C00675=1227.827,356.796,-73.722,-175.902,7.359,148.198
C00676=1227.832,356.549,-73.691,-175.904,7.356,148.197
C00677=1227.836,356.300,-73.658,-175.906,7.353,148.197
C00678=1227.840,356.052,-73.625,-175.908,7.351,148.197
C00679=1227.844,355.804,-73.593,-175.909,7.348,148.197
C00680=1227.849,355.557,-73.561,-175.910,7.345,148.196
C00681=1227.852,355.309,-73.529,-175.913,7.342,148.196
C00682=1227.857,355.061,-73.496,-175.914,7.339,148.196
C00683=1227.860,354.813,-73.465,-175.916,7.337,148.196
C00684=1227.865,354.565,-73.432,-175.917,7.334,148.196
C00685=1227.869,354.318,-73.400,-175.919,7.332,148.195
C00686=1227.873,354.070,-73.368,-175.921,7.328,148.195
C00687=1227.878,353.821,-73.335,-175.922,7.326,148.195
C00688=1227.881,353.573,-73.303,-175.924,7.323,148.195
C00689=1227.886,353.326,-73.270,-175.926,7.321,148.194
C00690=1227.890,353.078,-73.239,-175.927,7.318,148.194
C00691=1227.894,352.830,-73.206,-175.929,7.315,148.194
C00692=1227.898,352.582,-73.174,-175.931,7.312,148.194
C00693=1227.903,352.334,-73.142,-175.933,7.310,148.194
C00694=1227.906,352.087,-73.110,-175.934,7.307,148.193
C00695=1227.911,351.838,-73.077,-175.936,7.305,148.193
C00696=1227.915,351.591,-73.046,-175.938,7.301,148.193
C00697=1227.919,351.343,-73.014,-175.940,7.299,148.193
C00698=1227.923,351.095,-72.981,-175.941,7.296,148.193
C00699=1227.927,350.847,-72.950,-175.943,7.293,148.192
C00700=1227.932,350.599,-72.918,-175.945,7.290,148.192
C00701=1227.936,350.351,-72.886,-175.946,7.287,148.192
C00702=1227.940,350.103,-72.853,-175.948,7.285,148.192
C00703=1227.944,349.856,-72.821,-175.950,7.282,148.192
C00704=1227.949,349.607,-72.789,-175.951,7.280,148.191
C00705=1227.952,349.359,-72.757,-175.953,7.276,148.191
C00706=1227.957,349.112,-72.725,-175.955,7.274,148.191
C00707=1227.961,348.864,-72.693,-175.957,7.272,148.191
C00708=1227.965,348.616,-72.661,-175.959,7.269,148.191
C00709=1227.970,348.368,-72.629,-175.961,7.266,148.191
C00710=1227.974,348.120,-72.597,-175.963,7.263,148.190
C00711=1227.977,347.872,-72.565,-175.964,7.261,148.190
C00712=1227.982,347.624,-72.533,-175.966,7.258,148.190
C00713=1227.986,347.376,-72.501,-175.968,7.255,148.190
C00714=1227.990,347.128,-72.469,-175.970,7.252,148.190
C00715=1227.995,346.881,-72.437,-175.971,7.250,148.189
C00716=1227.999,346.633,-72.406,-175.973,7.247,148.189
C00717=1228.003,346.385,-72.374,-175.975,7.244,148.189
C00718=1228.008,346.136,-72.342,-175.977,7.241,148.189
C00719=1228.011,345.888,-72.311,-175.978,7.239,148.189
C00720=1228.016,345.641,-72.279,-175.980,7.237,148.189
C00721=1228.020,345.392,-72.247,-175.983,7.233,148.188
C00722=1228.024,345.144,-72.215,-175.984,7.231,148.188
C00723=1228.028,344.897,-72.183,-175.986,7.228,148.188
C00724=1228.033,344.649,-72.151,-175.987,7.226,148.188
C00725=1228.037,344.401,-72.119,-175.990,7.222,148.188
C00726=1228.041,344.153,-72.088,-175.991,7.220,148.187
C00727=1228.045,343.905,-72.056,-175.993,7.217,148.188
C00728=1228.050,343.657,-72.024,-175.995,7.215,148.187
C00729=1228.053,343.409,-71.992,-175.997,7.212,148.187
C00730=1228.058,343.162,-71.961,-175.999,7.209,148.187
C00731=1228.062,342.913,-71.930,-176.000,7.207,148.187
C00732=1228.067,342.665,-71.898,-176.003,7.203,148.187
C00733=1228.070,342.417,-71.866,-176.005,7.201,148.187
C00734=1228.074,342.169,-71.834,-176.006,7.198,148.186
C00735=1228.079,341.921,-71.803,-176.008,7.196,148.186
C00736=1228.084,341.644,-71.767,-176.011,7.193,148.186
C00737=1228.088,341.366,-71.731,-176.013,7.189,148.186
C00738=1228.093,341.089,-71.697,-176.014,7.187,148.186
C00739=1228.098,340.811,-71.661,-176.017,7.184,148.186
C00740=1228.101,340.563,-71.630,-176.019,7.181,148.186
C00741=1228.106,340.315,-71.599,-176.021,7.178,148.185
C00742=1228.110,340.067,-71.566,-176.022,7.175,148.185
C00743=1228.115,339.819,-71.535,-176.024,7.173,148.185
C00744=1228.119,339.571,-71.504,-176.026,7.171,148.185
C00745=1228.123,339.323,-71.472,-176.028,7.167,148.185
C00746=1228.127,339.075,-71.440,-176.030,7.165,148.185
C00747=1228.131,338.827,-71.410,-176.032,7.163,148.185
C00748=1228.135,338.579,-71.378,-176.034,7.159,148.184
C00749=1228.140,338.331,-71.347,-176.036,7.157,148.184
C00750=1228.144,338.083,-71.315,-176.038,7.154,148.184
C00751=1228.148,337.836,-71.283,-176.040,7.152,148.184
C00752=1228.152,337.587,-71.252,-176.042,7.149,148.184
C00753=1228.157,337.340,-71.220,-176.044,7.146,148.184
C00754=1228.161,337.091,-71.189,-176.045,7.144,148.184
C00755=1228.165,336.844,-71.158,-176.048,7.140,148.183
C00756=1228.169,336.595,-71.127,-176.050,7.138,148.184
C00757=1228.173,336.348,-71.095,-176.051,7.136,148.183
C00758=1228.177,336.099,-71.064,-176.054,7.133,148.183
C00759=1228.182,335.852,-71.033,-176.056,7.130,148.183
C00760=1228.186,335.603,-71.002,-176.057,7.128,148.183
C00761=1228.190,335.356,-70.970,-176.059,7.125,148.183
C00762=1228.194,335.107,-70.939,-176.062,7.122,148.183
C00763=1228.199,334.859,-70.908,-176.064,7.120,148.183
C00764=1228.203,334.612,-70.877,-176.065,7.117,148.183
C00765=1228.207,334.363,-70.846,-176.067,7.114,148.182
C00766=1228.211,334.116,-70.814,-176.070,7.112,148.182
C00767=1228.215,333.867,-70.783,-176.071,7.109,148.182
C00768=1228.220,333.620,-70.751,-176.074,7.106,148.182
C00769=1228.224,333.371,-70.720,-176.075,7.103,148.182
C00770=1228.228,333.123,-70.690,-176.078,7.101,148.182
C00771=1228.232,332.876,-70.658,-176.079,7.099,148.182
C00772=1228.237,332.627,-70.627,-176.082,7.096,148.182
C00773=1228.241,332.379,-70.596,-176.083,7.093,148.182
C00774=1228.245,332.131,-70.564,-176.086,7.091,148.182
C00775=1228.249,331.883,-70.534,-176.088,7.087,148.182
C00776=1228.254,331.635,-70.503,-176.090,7.085,148.182
C00777=1228.258,331.387,-70.472,-176.091,7.083,148.181
C00778=1228.262,331.139,-70.440,-176.094,7.080,148.181
C00779=1228.266,330.891,-70.409,-176.096,7.077,148.181
C00780=1228.270,330.643,-70.379,-176.098,7.075,148.181
C00781=1228.275,330.395,-70.348,-176.100,7.072,148.181
C00782=1228.279,330.147,-70.316,-176.102,7.069,148.181
C00783=1228.283,329.899,-70.286,-176.104,7.067,148.181
C00784=1228.288,329.651,-70.255,-176.106,7.065,148.181
C00785=1228.292,329.402,-70.224,-176.108,7.061,148.181
C00786=1228.296,329.154,-70.193,-176.110,7.059,148.181
C00787=1228.300,328.907,-70.162,-176.112,7.056,148.181
C00788=1228.304,328.659,-70.131,-176.114,7.053,148.181
C00789=1228.309,328.411,-70.100,-176.116,7.051,148.181
C00790=1228.313,328.162,-70.069,-176.118,7.049,148.180
C00791=1228.317,327.914,-70.038,-176.121,7.046,148.180
C00792=1228.322,327.666,-70.007,-176.122,7.043,148.180
C00793=1228.326,327.419,-69.977,-176.124,7.041,148.180
C00794=1228.329,327.170,-69.945,-176.127,7.038,148.180
C00795=1228.334,326.923,-69.915,-176.129,7.035,148.180
C00796=1228.339,326.675,-69.884,-176.131,7.033,148.180
C00797=1228.343,326.426,-69.853,-176.132,7.030,148.180
C00798=1228.347,326.178,-69.823,-176.135,7.027,148.180
C00799=1228.351,325.930,-69.792,-176.137,7.025,148.180
C00800=1228.355,325.682,-69.761,-176.139,7.023,148.180
C00801=1228.360,325.434,-69.730,-176.141,7.020,148.180
C00802=1228.364,325.186,-69.700,-176.144,7.017,148.180
C00803=1228.368,324.937,-69.669,-176.145,7.015,148.180
C00804=1228.372,324.689,-69.638,-176.148,7.012,148.180
C00805=1228.376,324.442,-69.608,-176.150,7.010,148.180
C00806=1228.381,324.194,-69.577,-176.152,7.007,148.180
C00807=1228.385,323.945,-69.546,-176.154,7.004,148.180
C00808=1228.389,323.697,-69.516,-176.156,7.002,148.180
C00809=1228.393,323.450,-69.485,-176.158,6.999,148.179
C00810=1228.398,323.202,-69.454,-176.161,6.996,148.179
C00811=1228.401,322.953,-69.424,-176.163,6.994,148.179
C00812=1228.406,322.705,-69.394,-176.165,6.992,148.180
C00813=1228.411,322.457,-69.363,-176.167,6.988,148.179
C00814=1228.415,322.209,-69.333,-176.169,6.986,148.179
C00815=1228.419,321.960,-69.301,-176.171,6.984,148.179
C00816=1228.423,321.712,-69.271,-176.173,6.981,148.179
C00817=1228.427,321.465,-69.241,-176.175,6.978,148.179
C00818=1228.432,321.217,-69.210,-176.178,6.976,148.179
C00819=1228.437,320.968,-69.180,-176.180,6.974,148.179
C00820=1228.440,320.720,-69.149,-176.182,6.970,148.179
C00821=1228.445,320.472,-69.118,-176.184,6.968,148.179
C00822=1228.448,320.224,-69.088,-176.186,6.966,148.179
C00823=1228.453,319.976,-69.057,-176.189,6.963,148.179
C00824=1228.457,319.728,-69.028,-176.190,6.960,148.179
C00825=1228.461,319.479,-68.997,-176.192,6.958,148.179
C00826=1228.466,319.231,-68.966,-176.195,6.955,148.179
C00827=1228.470,318.984,-68.936,-176.197,6.953,148.179
C00828=1228.475,318.735,-68.906,-176.199,6.951,148.179
C00829=1228.478,318.488,-68.876,-176.201,6.947,148.179
C00830=1228.482,318.239,-68.845,-176.204,6.945,148.179
C00831=1228.487,317.991,-68.815,-176.206,6.943,148.179
C00832=1228.491,317.743,-68.784,-176.208,6.941,148.179
C00833=1228.495,317.495,-68.754,-176.210,6.938,148.179
C00834=1228.500,317.246,-68.724,-176.213,6.935,148.179
C00835=1228.504,316.999,-68.694,-176.214,6.933,148.179
C00836=1228.509,316.751,-68.663,-176.217,6.930,148.179
C00837=1228.512,316.502,-68.633,-176.219,6.928,148.179
C00838=1228.517,316.254,-68.603,-176.221,6.925,148.179
C00839=1228.521,316.006,-68.573,-176.224,6.922,148.179
C00840=1228.526,315.730,-68.539,-176.226,6.920,148.179
C00841=1228.531,315.454,-68.506,-176.228,6.917,148.179
C00842=1228.535,315.179,-68.472,-176.231,6.914,148.179
C00843=1228.540,314.903,-68.439,-176.233,6.912,148.179
C00844=1228.544,314.655,-68.408,-176.235,6.908,148.179
C00845=1228.549,314.406,-68.379,-176.237,6.906,148.179
C00846=1228.553,314.158,-68.348,-176.240,6.904,148.179
C00847=1228.557,313.910,-68.319,-176.242,6.901,148.179
C00848=1228.561,313.663,-68.288,-176.244,6.899,148.179
C00849=1228.566,313.414,-68.258,-176.246,6.896,148.179
C00850=1228.570,313.166,-68.228,-176.248,6.894,148.179
C00851=1228.575,312.918,-68.198,-176.251,6.891,148.179
C00852=1228.579,312.670,-68.168,-176.253,6.889,148.179
C00853=1228.582,312.421,-68.138,-176.255,6.887,148.179
C00854=1228.587,312.173,-68.107,-176.258,6.884,148.179
C00855=1228.591,311.925,-68.078,-176.260,6.881,148.179
C00856=1228.595,311.677,-68.049,-176.262,6.879,148.179
C00857=1228.600,311.429,-68.018,-176.264,6.876,148.179
C00858=1228.604,311.180,-67.988,-176.266,6.874,148.179
C00859=1228.608,310.932,-67.959,-176.269,6.871,148.179
C00860=1228.613,310.684,-67.928,-176.271,6.868,148.179
C00861=1228.617,310.436,-67.899,-176.273,6.866,148.179
C00862=1228.621,310.188,-67.869,-176.275,6.864,148.179
C00863=1228.626,309.940,-67.838,-176.278,6.862,148.179
C00864=1228.630,309.691,-67.809,-176.280,6.859,148.179
C00865=1228.634,309.443,-67.780,-176.282,6.856,148.179
C00866=1228.638,309.195,-67.749,-176.284,6.854,148.179
C00867=1228.643,308.947,-67.719,-176.287,6.851,148.179
C00868=1228.647,308.699,-67.690,-176.289,6.849,148.180
C00869=1228.651,308.450,-67.660,-176.291,6.847,148.180
C00870=1228.655,308.203,-67.630,-176.293,6.844,148.180
C00871=1228.660,307.954,-67.600,-176.296,6.841,148.180
C00872=1228.664,307.706,-67.571,-176.298,6.839,148.180
C00873=1228.669,307.458,-67.541,-176.300,6.837,148.180
C00874=1228.673,307.210,-67.511,-176.303,6.834,148.180
C00875=1228.677,306.961,-67.481,-176.305,6.832,148.180
C00876=1228.682,306.713,-67.452,-176.307,6.829,148.180
C00877=1228.686,306.465,-67.422,-176.310,6.826,148.180
C00878=1228.690,306.217,-67.393,-176.312,6.824,148.180
C00879=1228.694,305.968,-67.363,-176.314,6.822,148.180
C00880=1228.700,305.720,-67.334,-176.316,6.820,148.180
C00881=1228.704,305.473,-67.303,-176.319,6.817,148.180
C00882=1228.708,305.225,-67.274,-176.321,6.815,148.180
C00883=1228.712,304.976,-67.245,-176.323,6.812,148.180
C00884=1228.716,304.728,-67.215,-176.326,6.809,148.180
C00885=1228.720,304.480,-67.186,-176.328,6.807,148.180
C00886=1228.724,304.231,-67.156,-176.330,6.805,148.180
C00887=1228.729,303.983,-67.126,-176.332,6.803,148.181
C00888=1228.734,303.735,-67.097,-176.335,6.800,148.181
C00889=1228.738,303.486,-67.067,-176.337,6.797,148.181
C00890=1228.742,303.238,-67.038,-176.339,6.795,148.181
C00891=1228.746,302.990,-67.008,-176.341,6.793,148.181
C00892=1228.751,302.742,-66.979,-176.344,6.790,148.181
C00893=1228.755,302.494,-66.950,-176.347,6.788,148.181
C00894=1228.759,302.246,-66.920,-176.349,6.786,148.181
C00895=1228.763,301.997,-66.891,-176.351,6.783,148.181
C00896=1228.768,301.749,-66.861,-176.353,6.781,148.181
C00897=1228.772,301.501,-66.832,-176.356,6.778,148.181
C00898=1228.776,301.253,-66.802,-176.358,6.776,148.181
C00899=1228.780,301.004,-66.773,-176.360,6.773,148.181
C00900=1228.785,300.756,-66.745,-176.362,6.771,148.181
C00901=1228.789,300.508,-66.715,-176.365,6.769,148.182
C00902=1228.794,300.260,-66.686,-176.367,6.767,148.182
C00903=1228.798,300.011,-66.656,-176.370,6.764,148.182
C00904=1228.802,299.763,-66.627,-176.372,6.761,148.182
C00905=1228.806,299.515,-66.597,-176.374,6.759,148.182
C00906=1228.811,299.267,-66.568,-176.377,6.756,148.182
C00907=1228.815,299.018,-66.540,-176.379,6.754,148.182
C00908=1228.820,298.770,-66.510,-176.381,6.752,148.182
C00909=1228.824,298.522,-66.481,-176.383,6.750,148.182
C00910=1228.828,298.274,-66.451,-176.386,6.747,148.182
C00911=1228.833,298.026,-66.422,-176.388,6.745,148.182
C00912=1228.837,297.777,-66.393,-176.391,6.743,148.182
C00913=1228.841,297.529,-66.364,-176.393,6.740,148.183
C00914=1228.846,297.281,-66.334,-176.396,6.737,148.183
C00915=1228.850,297.032,-66.305,-176.398,6.735,148.183
C00916=1228.855,296.784,-66.277,-176.400,6.733,148.183
C00917=1228.859,296.536,-66.247,-176.402,6.731,148.183
C00918=1228.863,296.288,-66.218,-176.405,6.728,148.183
C00919=1228.867,296.039,-66.190,-176.407,6.726,148.183
C00920=1228.871,295.791,-66.160,-176.409,6.724,148.183
C00921=1228.876,295.543,-66.131,-176.411,6.721,148.183
C00922=1228.880,295.294,-66.102,-176.414,6.719,148.183
C00923=1228.885,295.046,-66.073,-176.417,6.716,148.183
C00924=1228.889,294.798,-66.043,-176.419,6.714,148.183
C00925=1228.893,294.550,-66.016,-176.421,6.712,148.184
C00926=1228.897,294.302,-65.986,-176.424,6.709,148.184
C00927=1228.902,294.053,-65.957,-176.426,6.707,148.184
C00928=1228.906,293.804,-65.928,-176.428,6.705,148.184
C00929=1228.911,293.557,-65.899,-176.430,6.703,148.184
C00930=1228.915,293.308,-65.871,-176.433,6.700,148.184
C00931=1228.919,293.060,-65.841,-176.436,6.698,148.184
C00932=1228.924,292.812,-65.813,-176.438,6.695,148.184
C00933=1228.928,292.564,-65.783,-176.440,6.693,148.185
C00934=1228.932,292.315,-65.755,-176.443,6.690,148.185
C00935=1228.936,292.067,-65.726,-176.445,6.688,148.185
C00936=1228.941,291.819,-65.698,-176.447,6.686,148.185
C00937=1228.945,291.570,-65.668,-176.450,6.684,148.185
C00938=1228.950,291.321,-65.639,-176.452,6.682,148.185
C00939=1228.954,291.074,-65.611,-176.454,6.679,148.185
C00940=1228.958,290.825,-65.582,-176.457,6.677,148.185
C00941=1228.962,290.577,-65.553,-176.459,6.675,148.185
C00942=1228.967,290.329,-65.525,-176.461,6.672,148.185
C00943=1228.971,290.080,-65.496,-176.464,6.669,148.185
C00944=1228.976,289.807,-65.464,-176.467,6.667,148.186
C00945=1228.981,289.532,-65.432,-176.469,6.664,148.186
C00946=1228.985,289.258,-65.401,-176.472,6.663,148.186
C00947=1228.991,288.984,-65.369,-176.474,6.659,148.186
C00948=1228.994,288.736,-65.340,-176.477,6.658,148.186
C00949=1228.999,288.487,-65.312,-176.479,6.655,148.186
C00950=1229.004,288.239,-65.283,-176.482,6.652,148.186
C00951=1229.007,287.991,-65.254,-176.484,6.650,148.187
C00952=1229.012,287.743,-65.226,-176.486,6.648,148.187
C00953=1229.017,287.494,-65.197,-176.489,6.646,148.187
C00954=1229.021,287.245,-65.169,-176.491,6.644,148.187
C00955=1229.025,286.998,-65.140,-176.494,6.641,148.187
C00956=1229.030,286.749,-65.111,-176.496,6.639,148.187
C00957=1229.034,286.500,-65.083,-176.499,6.637,148.188
C00958=1229.039,286.252,-65.055,-176.501,6.635,148.188
C00959=1229.042,286.004,-65.026,-176.503,6.633,148.188
C00960=1229.047,285.756,-64.998,-176.506,6.630,148.188
C00961=1229.051,285.508,-64.969,-176.508,6.627,148.188
C00962=1229.056,285.259,-64.941,-176.511,6.626,148.188
C00963=1229.061,285.010,-64.912,-176.513,6.623,148.188
C00964=1229.064,284.763,-64.883,-176.515,6.621,148.188
C00965=1229.069,284.514,-64.855,-176.518,6.618,148.189
C00966=1229.073,284.266,-64.827,-176.520,6.616,148.189
C00967=1229.078,284.018,-64.799,-176.523,6.614,148.189
C00968=1229.082,283.769,-64.770,-176.525,6.612,148.189
C00969=1229.087,283.521,-64.742,-176.527,6.610,148.189
C00970=1229.090,283.272,-64.714,-176.530,6.607,148.189
C00971=1229.096,283.024,-64.686,-176.532,6.605,148.189
C00972=1229.099,282.775,-64.657,-176.535,6.603,148.190
C00973=1229.104,282.528,-64.628,-176.537,6.601,148.190
C00974=1229.108,282.279,-64.600,-176.539,6.599,148.190
C00975=1229.112,282.030,-64.571,-176.542,6.596,148.190
C00976=1229.117,281.783,-64.544,-176.544,6.594,148.190
C00977=1229.121,281.534,-64.515,-176.547,6.592,148.190
C00978=1229.126,281.286,-64.487,-176.549,6.590,148.190
C00979=1229.129,281.037,-64.459,-176.552,6.588,148.191
C00980=1229.134,280.789,-64.431,-176.554,6.585,148.191
C00981=1229.138,280.540,-64.402,-176.557,6.583,148.191
C00982=1229.143,280.292,-64.374,-176.559,6.580,148.191
C00983=1229.147,280.044,-64.346,-176.561,6.578,148.191
C00984=1229.151,279.796,-64.318,-176.564,6.576,148.191
C00985=1229.156,279.546,-64.290,-176.566,6.574,148.192
C00986=1229.160,279.298,-64.262,-176.568,6.572,148.192
C00987=1229.166,279.050,-64.234,-176.571,6.569,148.192
C00988=1229.169,278.802,-64.206,-176.574,6.567,148.192
C00989=1229.174,278.554,-64.178,-176.576,6.565,148.192
C00990=1229.178,278.305,-64.149,-176.578,6.563,148.193
C00991=1229.182,278.057,-64.122,-176.580,6.561,148.193
C00992=1229.186,277.808,-64.093,-176.583,6.559,148.193
C00993=1229.192,277.560,-64.066,-176.586,6.556,148.193
C00994=1229.195,277.311,-64.038,-176.588,6.554,148.193
C00995=1229.200,277.063,-64.010,-176.590,6.552,148.193
C00996=1229.204,276.814,-63.981,-176.593,6.550,148.194
C00997=1229.209,276.566,-63.953,-176.595,6.548,148.194
C00998=1229.213,276.319,-63.926,-176.598,6.546,148.194
C00999=1229.217,276.069,-63.898,-176.600,6.543,148.194
C01000=1229.222,275.821,-63.870,-176.603,6.541,148.194
C01001=1229.226,275.573,-63.842,-176.605,6.539,148.194
C01002=1229.230,275.325,-63.814,-176.608,6.537,148.195
C01003=1229.236,275.076,-63.786,-176.610,6.535,148.195
C01004=1229.239,274.827,-63.758,-176.612,6.533,148.195
C01005=1229.244,274.579,-63.730,-176.614,6.530,148.195
C01006=1229.248,274.330,-63.703,-176.618,6.528,148.195
C01007=1229.252,274.082,-63.675,-176.620,6.526,148.195
C01008=1229.257,273.834,-63.647,-176.622,6.524,148.196
C01009=1229.261,273.585,-63.619,-176.624,6.521,148.196
C01010=1229.266,273.337,-63.592,-176.627,6.520,148.196
C01011=1229.270,273.089,-63.564,-176.629,6.517,148.196
C01012=1229.275,272.840,-63.536,-176.632,6.515,148.196
C01013=1229.279,272.592,-63.508,-176.634,6.512,148.196
C01014=1229.283,272.344,-63.480,-176.637,6.510,148.197
C01015=1229.287,272.095,-63.453,-176.639,6.508,148.197
C01016=1229.292,271.847,-63.425,-176.642,6.506,148.197
C01017=1229.296,271.598,-63.398,-176.644,6.504,148.197
C01018=1229.300,271.350,-63.370,-176.646,6.502,148.197
C01019=1229.306,271.101,-63.342,-176.649,6.500,148.198
C01020=1229.310,270.853,-63.314,-176.651,6.498,148.198
C01021=1229.314,270.604,-63.287,-176.654,6.495,148.198
C01022=1229.318,270.356,-63.259,-176.656,6.493,148.198
C01023=1229.323,270.108,-63.232,-176.659,6.491,148.198
C01024=1229.327,269.859,-63.204,-176.662,6.489,148.199
C01025=1229.331,269.611,-63.177,-176.664,6.487,148.199
C01026=1229.336,269.363,-63.149,-176.666,6.485,148.199
C01027=1229.340,269.113,-63.122,-176.668,6.483,148.199
C01028=1229.345,268.865,-63.093,-176.671,6.481,148.199
C01029=1229.350,268.617,-63.066,-176.674,6.478,148.199
C01030=1229.354,268.369,-63.038,-176.676,6.476,148.200
C01031=1229.358,268.120,-63.011,-176.679,6.474,148.200
C01032=1229.363,267.871,-62.984,-176.681,6.472,148.200
C01033=1229.367,267.623,-62.956,-176.684,6.470,148.200
C01034=1229.372,267.375,-62.929,-176.686,6.468,148.201
C01035=1229.375,267.126,-62.901,-176.688,6.466,148.201
C01036=1229.380,266.878,-62.874,-176.691,6.464,148.201
C01037=1229.385,266.629,-62.847,-176.693,6.462,148.201
C01038=1229.389,266.381,-62.819,-176.696,6.460,148.201
C01039=1229.393,266.132,-62.792,-176.698,6.457,148.201
C01040=1229.398,265.884,-62.765,-176.701,6.455,148.202
C01041=1229.402,265.636,-62.737,-176.704,6.453,148.202
C01042=1229.407,265.387,-62.710,-176.706,6.451,148.202
C01043=1229.411,265.138,-62.682,-176.708,6.449,148.202
C01044=1229.415,264.890,-62.655,-176.711,6.447,148.203
C01045=1229.420,264.642,-62.627,-176.713,6.445,148.203
C01046=1229.424,264.393,-62.600,-176.716,6.443,148.203
C01047=1229.429,264.145,-62.573,-176.718,6.441,148.203
C01048=1229.433,263.872,-62.543,-176.721,6.438,148.203
C01049=1229.438,263.599,-62.514,-176.724,6.436,148.204
C01050=1229.443,263.327,-62.483,-176.726,6.435,148.204
C01051=1229.448,263.054,-62.454,-176.729,6.432,148.204
C01052=1229.452,262.806,-62.426,-176.731,6.430,148.204
C01053=1229.457,262.558,-62.399,-176.734,6.428,148.205
C01054=1229.461,262.309,-62.372,-176.737,6.426,148.205
C01055=1229.466,262.061,-62.345,-176.739,6.424,148.205
C01056=1229.470,261.811,-62.318,-176.741,6.422,148.205
C01057=1229.475,261.563,-62.291,-176.744,6.420,148.206
C01058=1229.479,261.315,-62.264,-176.746,6.418,148.206
C01059=1229.483,261.066,-62.237,-176.749,6.416,148.206
C01060=1229.488,260.818,-62.209,-176.751,6.414,148.206
C01061=1229.492,260.570,-62.182,-176.753,6.412,148.206
C01062=1229.497,260.321,-62.155,-176.756,6.410,148.207
C01063=1229.501,260.072,-62.128,-176.759,6.407,148.207
C01064=1229.505,259.824,-62.101,-176.761,6.405,148.207
C01065=1229.510,259.575,-62.074,-176.764,6.403,148.207
C01066=1229.514,259.327,-62.047,-176.766,6.401,148.208
C01067=1229.519,259.078,-62.020,-176.769,6.399,148.208
C01068=1229.524,258.830,-61.993,-176.771,6.397,148.208
C01069=1229.527,258.582,-61.967,-176.774,6.395,148.208
C01070=1229.532,258.333,-61.940,-176.776,6.393,148.208
C01071=1229.537,258.085,-61.913,-176.779,6.391,148.209
C01072=1229.541,257.836,-61.885,-176.781,6.389,148.209
C01073=1229.545,257.587,-61.859,-176.783,6.387,148.209
C01074=1229.549,257.339,-61.832,-176.786,6.385,148.209
C01075=1229.554,257.090,-61.805,-176.788,6.383,148.210
C01076=1229.558,256.842,-61.779,-176.791,6.381,148.210
C01077=1229.563,256.593,-61.752,-176.793,6.379,148.210
C01078=1229.568,256.345,-61.725,-176.796,6.377,148.210
C01079=1229.572,256.096,-61.698,-176.798,6.375,148.211
C01080=1229.576,255.848,-61.671,-176.801,6.373,148.211
C01081=1229.581,255.599,-61.644,-176.803,6.371,148.211
C01082=1229.586,255.351,-61.617,-176.806,6.369,148.211
C01083=1229.590,255.102,-61.591,-176.808,6.367,148.212
C01084=1229.594,254.854,-61.564,-176.810,6.365,148.212
C01085=1229.599,254.605,-61.537,-176.813,6.363,148.212
C01086=1229.603,254.357,-61.511,-176.816,6.361,148.212
C01087=1229.608,254.108,-61.484,-176.818,6.358,148.212
C01088=1229.613,253.859,-61.457,-176.821,6.356,148.213
C01089=1229.616,253.611,-61.431,-176.824,6.355,148.213
C01090=1229.621,253.363,-61.404,-176.826,6.353,148.213
C01091=1229.625,253.114,-61.377,-176.828,6.350,148.213
C01092=1229.630,252.865,-61.351,-176.831,6.349,148.214
C01093=1229.635,252.617,-61.324,-176.834,6.347,148.214
C01094=1229.639,252.369,-61.297,-176.836,6.345,148.214
C01095=1229.643,252.120,-61.270,-176.838,6.343,148.214
C01096=1229.647,251.871,-61.245,-176.841,6.341,148.215
C01097=1229.652,251.623,-61.218,-176.843,6.339,148.215
C01098=1229.656,251.375,-61.191,-176.846,6.337,148.215
C01099=1229.661,251.126,-61.165,-176.848,6.335,148.215
C01100=1229.666,250.877,-61.138,-176.851,6.333,148.216
C01101=1229.670,250.629,-61.111,-176.853,6.331,148.216
C01102=1229.675,250.380,-61.085,-176.856,6.329,148.216
C01103=1229.678,250.132,-61.058,-176.858,6.327,148.216
C01104=1229.683,249.882,-61.032,-176.861,6.325,148.217
C01105=1229.687,249.634,-61.006,-176.863,6.323,148.217
C01106=1229.692,249.386,-60.979,-176.866,6.321,148.217
C01107=1229.696,249.137,-60.953,-176.869,6.319,148.218
C01108=1229.701,248.889,-60.926,-176.871,6.317,148.218
C01109=1229.705,248.640,-60.900,-176.873,6.315,148.218
C01110=1229.710,248.391,-60.873,-176.876,6.313,148.218
C01111=1229.714,248.142,-60.847,-176.879,6.311,148.219
C01112=1229.719,247.894,-60.820,-176.881,6.309,148.219
C01113=1229.723,247.646,-60.795,-176.883,6.307,148.219
C01114=1229.727,247.398,-60.768,-176.886,6.306,148.219
C01115=1229.732,247.149,-60.742,-176.889,6.304,148.220
C01116=1229.736,246.900,-60.715,-176.891,6.302,148.220
C01117=1229.741,246.651,-60.689,-176.893,6.300,148.220
C01118=1229.745,246.403,-60.663,-176.896,6.298,148.220
C01119=1229.749,246.154,-60.637,-176.898,6.296,148.221
C01120=1229.754,245.905,-60.611,-176.901,6.295,148.221
C01121=1229.758,245.657,-60.584,-176.903,6.293,148.221
C01122=1229.764,245.409,-60.558,-176.905,6.291,148.222
C01123=1229.768,245.160,-60.532,-176.908,6.289,148.222
C01124=1229.772,244.912,-60.506,-176.910,6.287,148.222
C01125=1229.777,244.662,-60.480,-176.913,6.285,148.222
C01126=1229.781,244.414,-60.453,-176.916,6.283,148.223
C01127=1229.785,244.165,-60.427,-176.918,6.281,148.223
C01128=1229.790,243.916,-60.401,-176.920,6.279,148.223
C01129=1229.795,243.669,-60.375,-176.923,6.277,148.223
C01130=1229.799,243.420,-60.349,-176.926,6.275,148.224
C01131=1229.804,243.171,-60.323,-176.928,6.273,148.224
C01132=1229.808,242.923,-60.296,-176.931,6.272,148.224
C01133=1229.812,242.674,-60.271,-176.933,6.269,148.225
C01134=1229.817,242.425,-60.244,-176.936,6.267,148.225
C01135=1229.821,242.177,-60.218,-176.938,6.266,148.225
C01136=1229.826,241.929,-60.192,-176.941,6.264,148.225
C01137=1229.831,241.679,-60.166,-176.943,6.262,148.226
C01138=1229.835,241.431,-60.140,-176.946,6.260,148.226
C01139=1229.839,241.182,-60.115,-176.948,6.258,148.226
C01140=1229.844,240.934,-60.088,-176.951,6.256,148.226
C01141=1229.849,240.685,-60.062,-176.953,6.254,148.227
C01142=1229.853,240.436,-60.036,-176.956,6.252,148.227
C01143=1229.857,240.188,-60.011,-176.959,6.250,148.227
C01144=1229.862,239.939,-59.985,-176.961,6.249,148.228
C01145=1229.866,239.691,-59.958,-176.963,6.247,148.228
C01146=1229.871,239.442,-59.932,-176.966,6.245,148.228
C01147=1229.875,239.193,-59.907,-176.968,6.243,148.228
C01148=1229.880,238.945,-59.881,-176.971,6.241,148.229
C01149=1229.884,238.696,-59.855,-176.973,6.239,148.229
C01150=1229.889,238.447,-59.829,-176.976,6.238,148.229
C01151=1229.893,238.199,-59.803,-176.979,6.236,148.230
C01152=1229.898,237.928,-59.775,-176.981,6.234,148.230
C01153=1229.903,237.656,-59.747,-176.984,6.232,148.230
C01154=1229.908,237.385,-59.719,-176.987,6.229,148.231
C01155=1229.912,237.114,-59.691,-176.990,6.227,148.231
C01156=1229.917,236.865,-59.665,-176.992,6.225,148.231
C01157=1229.922,236.617,-59.639,-176.995,6.224,148.232
C01158=1229.926,236.368,-59.614,-176.997,6.222,148.232
C01159=1229.930,236.119,-59.588,-177.000,6.219,148.232
C01160=1229.936,235.871,-59.562,-177.002,6.218,148.232
C01161=1229.940,235.622,-59.536,-177.004,6.217,148.233
C01162=1229.944,235.373,-59.510,-177.007,6.215,148.233
C01163=1229.948,235.124,-59.485,-177.009,6.213,148.233
C01164=1229.953,234.876,-59.460,-177.012,6.211,148.234
C01165=1229.958,234.627,-59.434,-177.015,6.209,148.234
C01166=1229.962,234.378,-59.409,-177.017,6.207,148.234
C01167=1229.967,234.130,-59.383,-177.020,6.205,148.235
C01168=1229.971,233.881,-59.357,-177.022,6.203,148.235
C01169=1229.975,233.632,-59.332,-177.025,6.201,148.235
C01170=1229.980,233.384,-59.306,-177.027,6.199,148.235
C01171=1229.984,233.135,-59.280,-177.030,6.197,148.236
C01172=1229.988,232.886,-59.255,-177.032,6.196,148.236
C01173=1229.993,232.638,-59.230,-177.035,6.195,148.236
C01174=1229.998,232.389,-59.204,-177.037,6.193,148.237
C01175=1230.003,232.141,-59.179,-177.040,6.191,148.237
C01176=1230.007,231.892,-59.153,-177.042,6.189,148.237
C01177=1230.011,231.643,-59.127,-177.045,6.187,148.238
C01178=1230.016,231.395,-59.102,-177.048,6.185,148.238
C01179=1230.020,231.146,-59.077,-177.050,6.183,148.238
C01180=1230.025,230.897,-59.051,-177.052,6.181,148.238
C01181=1230.029,230.649,-59.026,-177.055,6.179,148.239
C01182=1230.034,230.400,-59.000,-177.057,6.178,148.239
C01183=1230.039,230.151,-58.975,-177.060,6.176,148.239
C01184=1230.043,229.902,-58.950,-177.062,6.174,148.240
C01185=1230.047,229.654,-58.924,-177.065,6.173,148.240
C01186=1230.052,229.406,-58.899,-177.068,6.171,148.240
C01187=1230.057,229.156,-58.874,-177.070,6.169,148.241
C01188=1230.061,228.908,-58.848,-177.073,6.167,148.241
C01189=1230.066,228.659,-58.822,-177.076,6.165,148.241
C01190=1230.071,228.410,-58.798,-177.078,6.163,148.242
C01191=1230.074,228.162,-58.773,-177.080,6.162,148.242
C01192=1230.078,227.913,-58.747,-177.083,6.160,148.242
C01193=1230.084,227.664,-58.722,-177.085,6.158,148.243
C01194=1230.088,227.416,-58.696,-177.088,6.157,148.243
C01195=1230.093,227.167,-58.672,-177.091,6.155,148.243
C01196=1230.097,226.918,-58.646,-177.093,6.153,148.243
C01197=1230.102,226.670,-58.621,-177.095,6.151,148.244
C01198=1230.106,226.421,-58.596,-177.098,6.149,148.244
C01199=1230.111,226.173,-58.571,-177.101,6.147,148.244
C01200=1230.115,225.923,-58.546,-177.103,6.146,148.245
C01201=1230.120,225.675,-58.520,-177.105,6.144,148.245
C01202=1230.125,225.426,-58.495,-177.108,6.142,148.245
C01203=1230.129,225.178,-58.471,-177.111,6.140,148.246
C01204=1230.133,224.929,-58.445,-177.113,6.138,148.246
C01205=1230.138,224.681,-58.420,-177.116,6.137,148.246
C01206=1230.142,224.431,-58.395,-177.118,6.135,148.247
C01207=1230.147,224.183,-58.370,-177.121,6.134,148.247
C01208=1230.151,223.934,-58.345,-177.123,6.132,148.247
C01209=1230.156,223.686,-58.320,-177.126,6.130,148.248
C01210=1230.160,223.436,-58.295,-177.128,6.128,148.248
C01211=1230.165,223.188,-58.269,-177.131,6.126,148.248
C01212=1230.169,222.939,-58.245,-177.134,6.124,148.249
C01213=1230.174,222.691,-58.220,-177.136,6.122,148.249
C01214=1230.178,222.442,-58.195,-177.139,6.121,148.249
C01215=1230.184,222.193,-58.170,-177.141,6.119,148.250
C01216=1230.187,221.944,-58.145,-177.144,6.118,148.250
C01217=1230.192,221.696,-58.120,-177.146,6.116,148.250
C01218=1230.197,221.446,-58.095,-177.149,6.114,148.251
C01219=1230.201,221.198,-58.070,-177.151,6.112,148.251
C01220=1230.206,220.950,-58.046,-177.154,6.110,148.251
C01221=1230.210,220.701,-58.020,-177.157,6.108,148.252
C01222=1230.215,220.453,-57.996,-177.159,6.107,148.252
C01223=1230.219,220.203,-57.971,-177.161,6.105,148.252
C01224=1230.224,219.954,-57.946,-177.164,6.104,148.253
C01225=1230.228,219.706,-57.921,-177.167,6.102,148.253
C01226=1230.233,219.457,-57.896,-177.169,6.100,148.253
C01227=1230.238,219.208,-57.872,-177.172,6.098,148.254
C01228=1230.241,218.960,-57.846,-177.174,6.097,148.254
C01229=1230.247,218.711,-57.822,-177.177,6.095,148.254
C01230=1230.250,218.462,-57.797,-177.179,6.093,148.255
C01231=1230.256,218.213,-57.773,-177.182,6.091,148.255
C01232=1230.261,217.965,-57.748,-177.185,6.089,148.255
C01233=1230.264,217.716,-57.723,-177.187,6.088,148.256
C01234=1230.269,217.467,-57.698,-177.190,6.086,148.256
C01235=1230.273,217.218,-57.674,-177.192,6.085,148.256
C01236=1230.278,216.970,-57.649,-177.194,6.083,148.257
C01237=1230.283,216.721,-57.625,-177.197,6.081,148.257
C01238=1230.287,216.472,-57.599,-177.200,6.079,148.257
C01239=1230.292,216.224,-57.575,-177.203,6.078,148.258
C01240=1230.296,215.975,-57.550,-177.205,6.076,148.258
C01241=1230.301,215.726,-57.525,-177.208,6.075,148.259
C01242=1230.305,215.477,-57.501,-177.210,6.073,148.259
C01243=1230.310,215.229,-57.477,-177.213,6.071,148.259
C01244=1230.314,214.980,-57.452,-177.215,6.069,148.260
C01245=1230.319,214.731,-57.428,-177.218,6.067,148.260
C01246=1230.324,214.482,-57.403,-177.221,6.065,148.260
C01247=1230.328,214.233,-57.378,-177.223,6.064,148.261
C01248=1230.333,213.985,-57.354,-177.225,6.062,148.261
C01249=1230.337,213.737,-57.329,-177.228,6.061,148.261
C01250=1230.341,213.487,-57.305,-177.231,6.059,148.262
C01251=1230.346,213.239,-57.280,-177.233,6.057,148.262
C01252=1230.351,212.990,-57.256,-177.235,6.056,148.262
C01253=1230.355,212.742,-57.232,-177.238,6.054,148.263
C01254=1230.360,212.492,-57.207,-177.241,6.052,148.263
C01255=1230.364,212.243,-57.183,-177.243,6.050,148.263
C01256=1230.370,211.973,-57.157,-177.246,6.049,148.264
C01257=1230.374,211.702,-57.130,-177.249,6.047,148.264
C01258=1230.379,211.432,-57.103,-177.252,6.045,148.264
C01259=1230.385,211.161,-57.077,-177.254,6.043,148.265
C01260=1230.389,210.913,-57.053,-177.257,6.042,148.265
C01261=1230.393,210.665,-57.029,-177.260,6.040,148.266
C01262=1230.398,210.415,-57.004,-177.263,6.038,148.266
C01263=1230.402,210.167,-56.980,-177.265,6.037,148.266
C01264=1230.407,209.918,-56.956,-177.267,6.035,148.267
C01265=1230.412,209.670,-56.931,-177.270,6.033,148.267
C01266=1230.416,209.420,-56.906,-177.273,6.031,148.267
C01267=1230.421,209.172,-56.882,-177.275,6.030,148.268
C01268=1230.426,208.923,-56.858,-177.277,6.028,148.268
C01269=1230.430,208.674,-56.834,-177.280,6.026,148.268
C01270=1230.434,208.425,-56.809,-177.283,6.025,148.269
C01271=1230.439,208.176,-56.785,-177.285,6.023,148.269
C01272=1230.443,207.928,-56.761,-177.288,6.022,148.270
C01273=1230.448,207.679,-56.738,-177.290,6.020,148.270
C01274=1230.453,207.430,-56.713,-177.293,6.018,148.270
C01275=1230.457,207.181,-56.689,-177.296,6.016,148.271
C01276=1230.461,206.933,-56.665,-177.298,6.015,148.271
C01277=1230.467,206.683,-56.641,-177.300,6.014,148.271
C01278=1230.471,206.435,-56.617,-177.303,6.012,148.272
C01279=1230.476,206.187,-56.592,-177.306,6.010,148.272
C01280=1230.480,205.938,-56.569,-177.308,6.008,148.272
C01281=1230.485,205.688,-56.544,-177.311,6.007,148.273
C01282=1230.489,205.440,-56.520,-177.313,6.005,148.273
C01283=1230.494,205.191,-56.496,-177.316,6.004,148.274
C01284=1230.498,204.942,-56.473,-177.319,6.002,148.274
C01285=1230.503,204.694,-56.448,-177.321,6.001,148.274
C01286=1230.508,204.445,-56.425,-177.323,5.999,148.275
C01287=1230.512,204.195,-56.400,-177.326,5.997,148.275
C01288=1230.516,203.947,-56.376,-177.329,5.995,148.275
C01289=1230.521,203.698,-56.353,-177.331,5.994,148.276
C01290=1230.526,203.449,-56.328,-177.334,5.993,148.276
C01291=1230.530,203.201,-56.304,-177.337,5.991,148.277
C01292=1230.535,202.952,-56.281,-177.339,5.989,148.277
C01293=1230.540,202.703,-56.256,-177.341,5.988,148.277
C01294=1230.544,202.454,-56.233,-177.344,5.986,148.278
C01295=1230.548,202.205,-56.209,-177.347,5.984,148.278
C01296=1230.553,201.956,-56.185,-177.349,5.982,148.278
C01297=1230.558,201.707,-56.161,-177.351,5.981,148.279
C01298=1230.563,201.458,-56.137,-177.354,5.980,148.279
C01299=1230.567,201.210,-56.113,-177.357,5.978,148.280
C01300=1230.572,200.961,-56.090,-177.360,5.976,148.280
C01301=1230.576,200.713,-56.066,-177.362,5.975,148.280
C01302=1230.581,200.464,-56.042,-177.364,5.973,148.281
C01303=1230.585,200.215,-56.018,-177.367,5.971,148.281
C01304=1230.590,199.966,-55.995,-177.370,5.969,148.281
C01305=1230.594,199.718,-55.971,-177.372,5.969,148.282
C01306=1230.599,199.468,-55.947,-177.375,5.967,148.282
C01307=1230.604,199.219,-55.923,-177.377,5.965,148.283
C01308=1230.608,198.970,-55.899,-177.380,5.964,148.283
C01309=1230.613,198.721,-55.876,-177.382,5.962,148.283
C01310=1230.617,198.473,-55.852,-177.385,5.960,148.284
C01311=1230.622,198.224,-55.828,-177.387,5.958,148.284
C01312=1230.626,197.975,-55.804,-177.390,5.958,148.285
C01313=1230.631,197.726,-55.781,-177.393,5.956,148.285
C01314=1230.636,197.477,-55.758,-177.395,5.954,148.285
C01315=1230.640,197.229,-55.734,-177.398,5.952,148.286
C01316=1230.645,196.980,-55.710,-177.400,5.951,148.286
C01317=1230.650,196.731,-55.687,-177.403,5.949,148.286
C01318=1230.654,196.482,-55.663,-177.406,5.948,148.287
C01319=1230.659,196.233,-55.639,-177.408,5.947,148.287
C01320=1230.663,195.984,-55.616,-177.410,5.945,148.288
C01321=1230.668,195.735,-55.593,-177.413,5.943,148.288
C01322=1230.672,195.487,-55.569,-177.415,5.942,148.288
C01323=1230.677,195.238,-55.545,-177.418,5.940,148.289
C01324=1230.682,194.989,-55.522,-177.421,5.939,148.289
C01325=1230.687,194.740,-55.498,-177.424,5.937,148.290
C01326=1230.691,194.491,-55.474,-177.426,5.936,148.290
C01327=1230.695,194.243,-55.452,-177.428,5.934,148.290
C01328=1230.700,193.994,-55.428,-177.431,5.932,148.291
C01329=1230.704,193.745,-55.405,-177.433,5.931,148.291
C01330=1230.709,193.496,-55.382,-177.436,5.930,148.292
C01331=1230.713,193.247,-55.357,-177.439,5.928,148.292
C01332=1230.718,192.998,-55.334,-177.441,5.927,148.292
C01333=1230.723,192.749,-55.311,-177.444,5.925,148.293
C01334=1230.728,192.501,-55.288,-177.446,5.923,148.293
C01335=1230.733,192.252,-55.264,-177.449,5.922,148.294
C01336=1230.737,192.003,-55.242,-177.451,5.920,148.294
C01337=1230.741,191.754,-55.218,-177.454,5.919,148.294
C01338=1230.746,191.506,-55.194,-177.456,5.918,148.295
C01339=1230.751,191.257,-55.171,-177.459,5.916,148.295
C01340=1230.755,191.007,-55.148,-177.462,5.914,148.296
C01341=1230.760,190.758,-55.124,-177.464,5.913,148.296
C01342=1230.765,190.509,-55.101,-177.467,5.911,148.296
C01343=1230.769,190.261,-55.078,-177.469,5.909,148.297
C01344=1230.773,190.012,-55.055,-177.471,5.908,148.297
C01345=1230.779,189.763,-55.032,-177.474,5.907,148.298
C01346=1230.783,189.514,-55.008,-177.477,5.905,148.298
C01347=1230.788,189.265,-54.985,-177.479,5.904,148.298
C01348=1230.792,189.017,-54.962,-177.482,5.902,148.299
C01349=1230.797,188.768,-54.939,-177.485,5.900,148.299
C01350=1230.801,188.518,-54.915,-177.487,5.900,148.300
C01351=1230.806,188.269,-54.892,-177.490,5.898,148.300
C01352=1230.810,188.021,-54.869,-177.492,5.896,148.300
C01353=1230.815,187.772,-54.846,-177.494,5.895,148.301
C01354=1230.820,187.523,-54.823,-177.498,5.893,148.301
C01355=1230.825,187.274,-54.800,-177.500,5.892,148.302
C01356=1230.829,187.026,-54.777,-177.502,5.891,148.302
C01357=1230.833,186.777,-54.754,-177.505,5.889,148.302
C01358=1230.838,186.527,-54.731,-177.508,5.887,148.303
C01359=1230.843,186.278,-54.708,-177.510,5.886,148.303
C01360=1230.848,186.008,-54.683,-177.513,5.884,148.304
C01361=1230.853,185.739,-54.657,-177.515,5.882,148.304
C01362=1230.858,185.470,-54.632,-177.519,5.881,148.305
C01363=1230.863,185.200,-54.608,-177.521,5.879,148.305
C01364=1230.867,184.951,-54.584,-177.524,5.878,148.306
C01365=1230.873,184.702,-54.562,-177.526,5.877,148.306
C01366=1230.877,184.453,-54.539,-177.529,5.875,148.306
C01367=1230.882,184.204,-54.516,-177.531,5.874,148.307
C01368=1230.886,183.956,-54.493,-177.534,5.872,148.307
C01369=1230.890,183.707,-54.470,-177.536,5.871,148.308
C01370=1230.896,183.458,-54.448,-177.539,5.869,148.308
C01371=1230.900,183.209,-54.425,-177.542,5.868,148.308
C01372=1230.905,182.960,-54.402,-177.544,5.867,148.309
C01373=1230.909,182.711,-54.378,-177.547,5.865,148.309
C01374=1230.914,182.461,-54.356,-177.550,5.863,148.310
C01375=1230.919,182.213,-54.333,-177.552,5.862,148.310
C01376=1230.923,181.964,-54.310,-177.554,5.860,148.310
C01377=1230.928,181.715,-54.288,-177.557,5.860,148.311
C01378=1230.932,181.466,-54.265,-177.560,5.858,148.311
C01379=1230.937,181.218,-54.242,-177.562,5.856,148.312
C01380=1230.942,180.969,-54.219,-177.564,5.855,148.312
C01381=1230.946,180.719,-54.197,-177.567,5.853,148.313
C01382=1230.951,180.470,-54.173,-177.569,5.852,148.313
C01383=1230.956,180.222,-54.152,-177.572,5.851,148.313
C01384=1230.960,179.973,-54.128,-177.575,5.849,148.314
C01385=1230.964,179.724,-54.105,-177.577,5.848,148.314
C01386=1230.970,179.475,-54.083,-177.580,5.846,148.315
C01387=1230.974,179.226,-54.060,-177.582,5.845,148.315
C01388=1230.979,178.977,-54.037,-177.585,5.844,148.316
C01389=1230.983,178.728,-54.015,-177.588,5.842,148.316
C01390=1230.988,178.480,-53.992,-177.590,5.841,148.316
C01391=1230.992,178.230,-53.970,-177.593,5.839,148.317
C01392=1230.997,177.981,-53.947,-177.595,5.838,148.317
C01393=1231.002,177.733,-53.925,-177.598,5.836,148.318
C01394=1231.007,177.484,-53.902,-177.601,5.835,148.318
C01395=1231.011,177.234,-53.879,-177.603,5.834,148.319
C01396=1231.016,176.986,-53.857,-177.606,5.832,148.319
C01397=1231.020,176.737,-53.834,-177.608,5.831,148.319
C01398=1231.025,176.487,-53.811,-177.610,5.829,148.320
C01399=1231.030,176.239,-53.789,-177.613,5.829,148.320
C01400=1231.034,175.990,-53.767,-177.616,5.827,148.321
C01401=1231.039,175.740,-53.744,-177.618,5.825,148.321
C01402=1231.044,175.492,-53.722,-177.621,5.824,148.322
C01403=1231.049,175.243,-53.699,-177.624,5.822,148.322
C01404=1231.053,174.994,-53.676,-177.626,5.821,148.323
C01405=1231.057,174.745,-53.655,-177.628,5.820,148.323
C01406=1231.062,174.496,-53.631,-177.631,5.819,148.323
C01407=1231.066,174.247,-53.609,-177.634,5.817,148.324
C01408=1231.072,173.998,-53.587,-177.636,5.815,148.324
C01409=1231.076,173.749,-53.564,-177.639,5.815,148.325
C01410=1231.081,173.501,-53.542,-177.641,5.813,148.325
C01411=1231.086,173.251,-53.520,-177.644,5.812,148.326
C01412=1231.090,173.002,-53.497,-177.647,5.810,148.326
C01413=1231.095,172.754,-53.475,-177.649,5.809,148.327
C01414=1231.100,172.504,-53.453,-177.651,5.807,148.327
C01415=1231.104,172.256,-53.430,-177.654,5.806,148.327
C01416=1231.108,172.007,-53.408,-177.657,5.805,148.328
C01417=1231.113,171.757,-53.386,-177.659,5.803,148.328
C01418=1231.118,171.509,-53.363,-177.661,5.802,148.329
C01419=1231.122,171.260,-53.341,-177.665,5.800,148.329
C01420=1231.128,171.011,-53.319,-177.667,5.799,148.330
C01421=1231.132,170.762,-53.296,-177.669,5.798,148.330
C01422=1231.136,170.513,-53.274,-177.672,5.797,148.331
C01423=1231.141,170.264,-53.252,-177.675,5.795,148.331
C01424=1231.146,170.014,-53.230,-177.677,5.794,148.331
C01425=1231.151,169.766,-53.208,-177.680,5.793,148.332
C01426=1231.155,169.517,-53.185,-177.682,5.792,148.332
C01427=1231.160,169.268,-53.164,-177.685,5.790,148.333
C01428=1231.165,169.019,-53.141,-177.687,5.789,148.333
C01429=1231.170,168.770,-53.119,-177.690,5.787,148.334
C01430=1231.174,168.521,-53.097,-177.692,5.785,148.334
C01431=1231.178,168.273,-53.075,-177.695,5.785,148.335
C01432=1231.183,168.023,-53.052,-177.698,5.783,148.335
C01433=1231.188,167.774,-53.030,-177.700,5.782,148.335
C01434=1231.193,167.525,-53.008,-177.703,5.780,148.336
C01435=1231.197,167.276,-52.987,-177.705,5.779,148.336
C01436=1231.202,167.027,-52.965,-177.708,5.778,148.337
C01437=1231.207,166.778,-52.943,-177.710,5.777,148.337
C01438=1231.211,166.529,-52.920,-177.713,5.775,148.338
C01439=1231.216,166.281,-52.898,-177.715,5.774,148.338
C01440=1231.220,166.031,-52.876,-177.718,5.773,148.339
C01441=1231.225,165.783,-52.854,-177.720,5.772,148.339
C01442=1231.230,165.533,-52.832,-177.723,5.770,148.339
C01443=1231.234,165.285,-52.811,-177.725,5.769,148.340
C01444=1231.239,165.036,-52.788,-177.728,5.767,148.340
C01445=1231.244,164.787,-52.766,-177.730,5.766,148.341
C01446=1231.249,164.537,-52.744,-177.733,5.765,148.341
C01447=1231.253,164.289,-52.722,-177.735,5.764,148.342
C01448=1231.258,164.039,-52.700,-177.739,5.762,148.342
C01449=1231.263,163.791,-52.679,-177.741,5.761,148.343
C01450=1231.267,163.541,-52.657,-177.743,5.759,148.343
C01451=1231.272,163.293,-52.635,-177.746,5.759,148.344
C01452=1231.276,163.043,-52.613,-177.749,5.757,148.344
C01453=1231.281,162.795,-52.591,-177.751,5.756,148.344
C01454=1231.286,162.546,-52.570,-177.754,5.754,148.345
C01455=1231.290,162.297,-52.548,-177.756,5.753,148.345
C01456=1231.296,162.048,-52.525,-177.759,5.752,148.346
C01457=1231.300,161.798,-52.504,-177.761,5.751,148.346
C01458=1231.305,161.549,-52.482,-177.764,5.749,148.347
C01459=1231.309,161.300,-52.460,-177.766,5.748,148.347
C01460=1231.314,161.051,-52.439,-177.769,5.747,148.348
C01461=1231.319,160.802,-52.417,-177.771,5.746,148.348
C01462=1231.323,160.553,-52.395,-177.774,5.744,148.349
C01463=1231.328,160.305,-52.373,-177.776,5.743,148.349
C01464=1231.333,160.035,-52.350,-177.780,5.742,148.350
C01465=1231.338,159.767,-52.326,-177.782,5.741,148.350
C01466=1231.344,159.497,-52.303,-177.785,5.739,148.351
C01467=1231.348,159.228,-52.280,-177.787,5.737,148.351
C01468=1231.353,158.979,-52.258,-177.790,5.737,148.352
C01469=1231.357,158.730,-52.236,-177.793,5.735,148.352
C01470=1231.362,158.481,-52.214,-177.795,5.734,148.353
C01471=1231.367,158.232,-52.193,-177.798,5.732,148.353
C01472=1231.372,157.983,-52.172,-177.800,5.731,148.353
C01473=1231.376,157.734,-52.150,-177.803,5.730,148.354
C01474=1231.381,157.485,-52.128,-177.805,5.729,148.354
C01475=1231.386,157.236,-52.107,-177.808,5.728,148.355
C01476=1231.390,156.986,-52.085,-177.811,5.726,148.355
C01477=1231.395,156.738,-52.063,-177.813,5.725,148.356
C01478=1231.400,156.489,-52.042,-177.816,5.724,148.356
C01479=1231.404,156.240,-52.021,-177.818,5.723,148.357
C01480=1231.409,155.991,-51.999,-177.821,5.721,148.357
C01481=1231.414,155.742,-51.978,-177.823,5.720,148.358
C01482=1231.418,155.492,-51.956,-177.826,5.718,148.358
C01483=1231.423,155.244,-51.934,-177.828,5.718,148.359
C01484=1231.428,154.994,-51.914,-177.831,5.716,148.359
C01485=1231.433,154.745,-51.891,-177.834,5.715,148.360
C01486=1231.437,154.496,-51.870,-177.836,5.714,148.360
C01487=1231.442,154.247,-51.849,-177.838,5.713,148.361
C01488=1231.447,153.999,-51.828,-177.841,5.712,148.361
C01489=1231.451,153.750,-51.806,-177.844,5.710,148.362
C01490=1231.456,153.500,-51.785,-177.846,5.709,148.362
C01491=1231.461,153.252,-51.763,-177.849,5.708,148.363
C01492=1231.466,153.002,-51.742,-177.852,5.707,148.363
C01493=1231.470,152.753,-51.721,-177.854,5.706,148.364
C01494=1231.475,152.504,-51.700,-177.856,5.704,148.364
C01495=1231.480,152.255,-51.678,-177.859,5.703,148.365
C01496=1231.484,152.005,-51.657,-177.862,5.702,148.365
C01497=1231.489,151.757,-51.635,-177.864,5.701,148.366
C01498=1231.493,151.508,-51.614,-177.867,5.699,148.366
C01499=1231.499,151.259,-51.593,-177.869,5.698,148.367
C01500=1231.503,151.009,-51.572,-177.872,5.697,148.367
C01501=1231.508,150.761,-51.550,-177.874,5.696,148.367
C01502=1231.512,150.512,-51.530,-177.877,5.695,148.368
C01503=1231.517,150.263,-51.508,-177.879,5.693,148.368
C01504=1231.522,150.013,-51.486,-177.882,5.692,148.369
C01505=1231.527,149.764,-51.465,-177.885,5.691,148.369
C01506=1231.531,149.515,-51.444,-177.887,5.690,148.370
C01507=1231.536,149.267,-51.423,-177.889,5.689,148.370
C01508=1231.541,149.018,-51.402,-177.893,5.688,148.371
C01509=1231.545,148.768,-51.381,-177.895,5.687,148.371
C01510=1231.550,148.519,-51.359,-177.897,5.685,148.372
C01511=1231.555,148.270,-51.338,-177.900,5.684,148.372
C01512=1231.559,148.022,-51.317,-177.902,5.683,148.373
C01513=1231.564,147.772,-51.296,-177.905,5.682,148.373
C01514=1231.569,147.522,-51.275,-177.907,5.681,148.374
C01515=1231.573,147.274,-51.254,-177.910,5.679,148.374
C01516=1231.578,147.025,-51.233,-177.913,5.678,148.375
C01517=1231.583,146.776,-51.212,-177.915,5.677,148.375
C01518=1231.588,146.527,-51.191,-177.918,5.676,148.376
C01519=1231.593,146.278,-51.170,-177.920,5.675,148.376
C01520=1231.597,146.028,-51.149,-177.923,5.673,148.377
C01521=1231.601,145.780,-51.128,-177.925,5.672,148.377
C01522=1231.607,145.530,-51.107,-177.928,5.672,148.378
C01523=1231.612,145.281,-51.086,-177.930,5.670,148.378
C01524=1231.616,145.032,-51.065,-177.933,5.669,148.379
C01525=1231.621,144.784,-51.044,-177.935,5.668,148.379
C01526=1231.626,144.535,-51.023,-177.938,5.667,148.380
C01527=1231.630,144.285,-51.002,-177.940,5.666,148.380
C01528=1231.635,144.036,-50.981,-177.944,5.664,148.381
C01529=1231.639,143.787,-50.960,-177.946,5.663,148.381
C01530=1231.645,143.538,-50.939,-177.948,5.662,148.382
C01531=1231.649,143.289,-50.918,-177.951,5.661,148.382
C01532=1231.654,143.040,-50.897,-177.954,5.660,148.383
C01533=1231.659,142.791,-50.877,-177.956,5.659,148.383
C01534=1231.664,142.542,-50.855,-177.959,5.658,148.384
C01535=1231.667,142.292,-50.835,-177.961,5.657,148.384
C01536=1231.673,142.043,-50.814,-177.964,5.655,148.385
C01537=1231.677,141.794,-50.793,-177.966,5.654,148.385
C01538=1231.682,141.545,-50.772,-177.969,5.653,148.386
C01539=1231.687,141.296,-50.752,-177.971,5.652,148.386
C01540=1231.692,141.047,-50.731,-177.974,5.651,148.387
C01541=1231.696,140.798,-50.711,-177.976,5.650,148.387
C01542=1231.701,140.549,-50.689,-177.979,5.648,148.388
C01543=1231.706,140.300,-50.669,-177.981,5.648,148.388
C01544=1231.711,140.051,-50.648,-177.984,5.647,148.389
C01545=1231.715,139.802,-50.627,-177.987,5.645,148.389
C01546=1231.720,139.553,-50.606,-177.989,5.644,148.390
C01547=1231.725,139.304,-50.586,-177.992,5.643,148.390
C01548=1231.730,139.055,-50.565,-177.995,5.642,148.391
C01549=1231.734,138.806,-50.545,-177.997,5.641,148.391
C01550=1231.739,138.556,-50.523,-178.000,5.639,148.392
C01551=1231.743,138.307,-50.503,-178.002,5.638,148.392
C01552=1231.748,138.058,-50.483,-178.004,5.638,148.393
C01553=1231.753,137.808,-50.462,-178.007,5.636,148.393
C01554=1231.757,137.560,-50.441,-178.010,5.635,148.394
C01555=1231.763,137.310,-50.420,-178.012,5.634,148.394
C01556=1231.767,137.061,-50.400,-178.015,5.633,148.395
C01557=1231.771,136.812,-50.379,-178.017,5.632,148.395
C01558=1231.777,136.563,-50.358,-178.020,5.631,148.396
C01559=1231.781,136.314,-50.338,-178.022,5.629,148.396
C01560=1231.786,136.065,-50.317,-178.025,5.629,148.397
C01561=1231.791,135.815,-50.298,-178.027,5.628,148.397
C01562=1231.795,135.566,-50.277,-178.030,5.626,148.398
C01563=1231.801,135.317,-50.256,-178.032,5.625,148.398
C01564=1231.805,135.068,-50.236,-178.035,5.625,148.399
C01565=1231.809,134.819,-50.215,-178.038,5.623,148.399
C01566=1231.815,134.570,-50.194,-178.040,5.622,148.400
C01567=1231.819,134.321,-50.174,-178.042,5.621,148.400
C01568=1231.825,134.052,-50.152,-178.046,5.620,148.401
C01569=1231.829,133.784,-50.131,-178.048,5.619,148.402
C01570=1231.835,133.516,-50.108,-178.051,5.618,148.402
C01571=1231.840,133.246,-50.086,-178.053,5.617,148.403
C01572=1231.845,132.998,-50.066,-178.057,5.615,148.403
C01573=1231.849,132.749,-50.046,-178.059,5.614,148.404
C01574=1231.855,132.499,-50.026,-178.061,5.614,148.404
C01575=1231.859,132.250,-50.005,-178.064,5.612,148.405
C01576=1231.864,132.001,-49.985,-178.067,5.611,148.405
C01577=1231.869,131.752,-49.964,-178.069,5.611,148.406
C01578=1231.873,131.503,-49.943,-178.071,5.610,148.406
C01579=1231.878,131.253,-49.924,-178.074,5.608,148.407
C01580=1231.882,131.004,-49.903,-178.077,5.607,148.407
C01581=1231.888,130.755,-49.882,-178.079,5.606,148.408
C01582=1231.892,130.505,-49.863,-178.082,5.605,148.408
C01583=1231.897,130.257,-49.842,-178.084,5.604,148.409
C01584=1231.902,130.008,-49.822,-178.087,5.603,148.409
C01585=1231.906,129.759,-49.802,-178.090,5.602,148.410
C01586=1231.912,129.509,-49.782,-178.092,5.601,148.411
C01587=1231.916,129.261,-49.761,-178.094,5.600,148.411
C01588=1231.921,129.012,-49.741,-178.097,5.599,148.412
C01589=1231.925,128.762,-49.721,-178.100,5.597,148.412
C01590=1231.930,128.513,-49.701,-178.102,5.597,148.413
C01591=1231.934,128.263,-49.681,-178.104,5.596,148.413
C01592=1231.940,128.014,-49.660,-178.108,5.594,148.414
C01593=1231.945,127.766,-49.640,-178.110,5.593,148.414
C01594=1231.949,127.516,-49.621,-178.112,5.593,148.415
C01595=1231.954,127.267,-49.600,-178.115,5.592,148.415
C01596=1231.959,127.018,-49.581,-178.118,5.590,148.416
C01597=1231.963,126.769,-49.560,-178.120,5.590,148.416
C01598=1231.967,126.520,-49.540,-178.122,5.589,148.417
C01599=1231.973,126.270,-49.520,-178.125,5.587,148.418
C01600=1231.978,126.022,-49.500,-178.128,5.586,148.418
C01601=1231.983,125.772,-49.480,-178.130,5.586,148.419
C01602=1231.987,125.523,-49.460,-178.133,5.585,148.419
C01603=1231.992,125.274,-49.440,-178.135,5.583,148.420
C01604=1231.996,125.025,-49.420,-178.138,5.583,148.420
C01605=1232.002,124.776,-49.400,-178.140,5.582,148.421
C01606=1232.006,124.527,-49.380,-178.143,5.581,148.421
C01607=1232.011,124.277,-49.360,-178.145,5.579,148.422
C01608=1232.015,124.029,-49.340,-178.148,5.579,148.422
C01609=1232.020,123.779,-49.320,-178.151,5.578,148.423
C01610=1232.026,123.530,-49.300,-178.153,5.577,148.423
C01611=1232.031,123.281,-49.280,-178.156,5.575,148.424
C01612=1232.035,123.032,-49.260,-178.158,5.574,148.424
C01613=1232.040,122.782,-49.240,-178.161,5.574,148.425
C01614=1232.045,122.533,-49.220,-178.164,5.572,148.426
C01615=1232.050,122.284,-49.200,-178.166,5.571,148.426
C01616=1232.054,122.035,-49.181,-178.169,5.571,148.427
C01617=1232.059,121.786,-49.160,-178.171,5.570,148.427
C01618=1232.063,121.536,-49.141,-178.174,5.568,148.428
C01619=1232.069,121.288,-49.121,-178.176,5.568,148.428
C01620=1232.073,121.039,-49.101,-178.179,5.567,148.429
C01621=1232.078,120.789,-49.081,-178.181,5.566,148.429
C01622=1232.083,120.539,-49.062,-178.183,5.565,148.430
C01623=1232.088,120.291,-49.042,-178.186,5.564,148.430
C01624=1232.093,120.042,-49.022,-178.189,5.563,148.431
C01625=1232.097,119.792,-49.002,-178.191,5.562,148.431
C01626=1232.101,119.543,-48.983,-178.194,5.561,148.432
C01627=1232.106,119.295,-48.963,-178.196,5.560,148.432
C01628=1232.111,119.045,-48.944,-178.199,5.559,148.433
C01629=1232.115,118.796,-48.923,-178.202,5.558,148.434
C01630=1232.120,118.546,-48.904,-178.204,5.557,148.434
C01631=1232.126,118.298,-48.884,-178.207,5.556,148.435
C01632=1232.130,118.048,-48.865,-178.209,5.555,148.435
C01633=1232.135,117.799,-48.844,-178.212,5.554,148.436
C01634=1232.140,117.550,-48.825,-178.214,5.554,148.436
C01635=1232.145,117.301,-48.805,-178.217,5.552,148.437
C01636=1232.150,117.051,-48.786,-178.220,5.551,148.438
C01637=1232.155,116.802,-48.766,-178.222,5.551,148.438
C01638=1232.159,116.554,-48.747,-178.224,5.550,148.439
C01639=1232.163,116.304,-48.727,-178.227,5.549,148.439
C01640=1232.169,116.055,-48.708,-178.230,5.547,148.440
C01641=1232.173,115.806,-48.688,-178.232,5.547,148.440
C01642=1232.178,115.556,-48.668,-178.235,5.546,148.441
C01643=1232.183,115.308,-48.648,-178.237,5.545,148.441
C01644=1232.188,115.058,-48.629,-178.240,5.544,148.442
C01645=1232.192,114.809,-48.610,-178.243,5.543,148.443
C01646=1232.197,114.560,-48.590,-178.245,5.542,148.443
C01647=1232.202,114.310,-48.571,-178.248,5.541,148.444
C01648=1232.207,114.061,-48.551,-178.250,5.540,148.444
C01649=1232.212,113.812,-48.532,-178.253,5.539,148.445
C01650=1232.217,113.562,-48.512,-178.255,5.538,148.445
C01651=1232.221,113.313,-48.493,-178.258,5.537,148.446
C01652=1232.226,113.064,-48.474,-178.260,5.537,148.446
C01653=1232.231,112.815,-48.453,-178.263,5.536,148.447
C01654=1232.236,112.567,-48.434,-178.265,5.534,148.447
C01655=1232.240,112.317,-48.415,-178.268,5.534,148.448
C01656=1232.245,112.068,-48.395,-178.271,5.533,148.449
C01657=1232.250,111.819,-48.376,-178.273,5.532,148.449
C01658=1232.255,111.569,-48.356,-178.275,5.531,148.450
C01659=1232.259,111.321,-48.338,-178.279,5.530,148.450
C01660=1232.264,111.071,-48.318,-178.281,5.529,148.451
C01661=1232.269,110.822,-48.298,-178.283,5.528,148.451
C01662=1232.274,110.573,-48.279,-178.286,5.528,148.452
C01663=1232.278,110.323,-48.260,-178.288,5.527,148.452
C01664=1232.284,110.075,-48.241,-178.291,5.526,148.453
C01665=1232.288,109.825,-48.221,-178.294,5.525,148.454
C01666=1232.292,109.576,-48.202,-178.296,5.524,148.454
C01667=1232.298,109.326,-48.183,-178.299,5.523,148.455
C01668=1232.303,109.077,-48.164,-178.301,5.522,148.455
C01669=1232.308,108.828,-48.145,-178.303,5.521,148.456
C01670=1232.312,108.579,-48.125,-178.306,5.520,148.456
C01671=1232.317,108.330,-48.106,-178.309,5.519,148.457
C01672=1232.322,108.061,-48.085,-178.311,5.518,148.458
C01673=1232.327,107.792,-48.064,-178.314,5.518,148.458
C01674=1232.333,107.524,-48.044,-178.317,5.516,148.459
C01675=1232.337,107.256,-48.024,-178.320,5.516,148.459
C01676=1232.343,107.007,-48.004,-178.322,5.515,148.460
C01677=1232.347,106.757,-47.985,-178.324,5.514,148.461
C01678=1232.352,106.509,-47.966,-178.328,5.513,148.461
C01679=1232.357,106.258,-47.947,-178.330,5.512,148.462
C01680=1232.362,106.009,-47.928,-178.332,5.511,148.462
C01681=1232.366,105.760,-47.909,-178.335,5.510,148.463
C01682=1232.372,105.511,-47.889,-178.337,5.510,148.463
C01683=1232.376,105.262,-47.870,-178.340,5.509,148.464
C01684=1232.381,105.013,-47.852,-178.343,5.507,148.465
C01685=1232.386,104.763,-47.832,-178.345,5.507,148.465
C01686=1232.391,104.514,-47.813,-178.348,5.506,148.466
C01687=1232.395,104.265,-47.794,-178.350,5.505,148.466
C01688=1232.400,104.016,-47.775,-178.353,5.505,148.467
C01689=1232.405,103.766,-47.756,-178.355,5.504,148.467
C01690=1232.410,103.518,-47.737,-178.358,5.502,148.468
C01691=1232.414,103.268,-47.718,-178.361,5.502,148.469
C01692=1232.419,103.019,-47.700,-178.363,5.501,148.469
C01693=1232.424,102.769,-47.680,-178.365,5.500,148.470
C01694=1232.429,102.520,-47.661,-178.368,5.499,148.470
C01695=1232.434,102.271,-47.642,-178.371,5.499,148.471
C01696=1232.439,102.022,-47.623,-178.373,5.498,148.471
C01697=1232.444,101.773,-47.604,-178.376,5.496,148.472
C01698=1232.449,101.523,-47.585,-178.379,5.496,148.473
C01699=1232.453,101.274,-47.567,-178.381,5.495,148.473
C01700=1232.458,101.025,-47.547,-178.383,5.494,148.474
C01701=1232.463,100.776,-47.529,-178.386,5.494,148.474
C01702=1232.467,100.526,-47.510,-178.389,5.493,148.475
C01703=1232.472,100.278,-47.491,-178.391,5.492,148.475
C01704=1232.477,100.028,-47.473,-178.393,5.491,148.476
C01705=1232.482,99.779,-47.453,-178.396,5.490,148.477
C01706=1232.487,99.530,-47.435,-178.399,5.489,148.477
C01707=1232.492,99.280,-47.416,-178.401,5.488,148.478
C01708=1232.496,99.031,-47.397,-178.404,5.488,148.478
C01709=1232.502,98.782,-47.378,-178.406,5.487,148.479
C01710=1232.506,98.533,-47.359,-178.409,5.486,148.479
C01711=1232.512,98.283,-47.341,-178.411,5.486,148.480
C01712=1232.516,98.034,-47.322,-178.414,5.484,148.481
C01713=1232.521,97.785,-47.304,-178.416,5.483,148.481
C01714=1232.526,97.536,-47.284,-178.419,5.482,148.482
C01715=1232.530,97.286,-47.266,-178.422,5.482,148.482
C01716=1232.536,97.037,-47.247,-178.424,5.481,148.483
C01717=1232.540,96.787,-47.228,-178.426,5.480,148.484
C01718=1232.544,96.539,-47.210,-178.429,5.480,148.484
C01719=1232.550,96.289,-47.191,-178.432,5.479,148.485
C01720=1232.554,96.040,-47.172,-178.434,5.478,148.485
C01721=1232.559,95.791,-47.154,-178.437,5.477,148.486
C01722=1232.564,95.542,-47.135,-178.440,5.476,148.487
C01723=1232.569,95.292,-47.116,-178.442,5.475,148.487
C01724=1232.574,95.043,-47.098,-178.444,5.474,148.488
C01725=1232.579,94.794,-47.079,-178.447,5.474,148.488
C01726=1232.583,94.544,-47.061,-178.450,5.473,148.489
C01727=1232.588,94.296,-47.042,-178.452,5.472,148.489
C01728=1232.594,94.046,-47.023,-178.454,5.472,148.490
C01729=1232.598,93.796,-47.005,-178.457,5.471,148.491
C01730=1232.602,93.548,-46.986,-178.460,5.470,148.491
C01731=1232.608,93.298,-46.968,-178.462,5.469,148.492
C01732=1232.612,93.049,-46.949,-178.465,5.468,148.492
C01733=1232.617,92.800,-46.931,-178.468,5.467,148.493
C01734=1232.623,92.550,-46.912,-178.470,5.467,148.494
C01735=1232.627,92.301,-46.893,-178.472,5.466,148.494
C01736=1232.632,92.052,-46.875,-178.475,5.465,148.495
C01737=1232.636,91.803,-46.857,-178.478,5.465,148.495
C01738=1232.642,91.553,-46.839,-178.480,5.464,148.496
C01739=1232.646,91.304,-46.820,-178.482,5.463,148.496
C01740=1232.651,91.055,-46.802,-178.485,5.463,148.497
C01741=1232.656,90.806,-46.784,-178.488,5.462,148.498
C01742=1232.661,90.556,-46.764,-178.491,5.460,148.498
C01743=1232.666,90.307,-46.746,-178.493,5.460,148.499
C01744=1232.671,90.058,-46.728,-178.495,5.459,148.499
C01745=1232.675,89.809,-46.710,-178.498,5.458,148.500
C01746=1232.679,89.559,-46.691,-178.501,5.458,148.501
C01747=1232.685,89.310,-46.672,-178.503,5.457,148.501
C01748=1232.690,89.061,-46.654,-178.505,5.456,148.502
C01749=1232.695,88.811,-46.636,-178.508,5.456,148.503
C01750=1232.699,88.562,-46.618,-178.511,5.455,148.503
C01751=1232.704,88.313,-46.599,-178.513,5.454,148.504
C01752=1232.709,88.063,-46.581,-178.515,5.453,148.504
C01753=1232.714,87.814,-46.563,-178.518,5.453,148.505
C01754=1232.719,87.564,-46.544,-178.521,5.452,148.506
C01755=1232.724,87.315,-46.526,-178.523,5.450,148.506
C01756=1232.729,87.066,-46.509,-178.526,5.450,148.507
C01757=1232.733,86.818,-46.490,-178.529,5.449,148.507
C01758=1232.739,86.568,-46.471,-178.531,5.449,148.508
C01759=1232.743,86.318,-46.453,-178.534,5.448,148.509
C01760=1232.748,86.069,-46.435,-178.536,5.447,148.509
C01761=1232.753,85.820,-46.417,-178.539,5.446,148.510
C01762=1232.758,85.571,-46.399,-178.541,5.446,148.510
C01763=1232.763,85.321,-46.381,-178.544,5.445,148.511
C01764=1232.767,85.072,-46.363,-178.546,5.444,148.511
C01765=1232.772,84.822,-46.345,-178.549,5.444,148.512
C01766=1232.777,84.573,-46.327,-178.551,5.443,148.513
C01767=1232.783,84.324,-46.308,-178.554,5.442,148.513
C01768=1232.787,84.075,-46.289,-178.556,5.442,148.514
C01769=1232.791,83.825,-46.271,-178.559,5.441,148.514
C01770=1232.796,83.576,-46.253,-178.561,5.440,148.515
C01771=1232.801,83.327,-46.235,-178.564,5.440,148.516
C01772=1232.806,83.078,-46.217,-178.566,5.439,148.516
C01773=1232.811,82.829,-46.199,-178.569,5.437,148.517
C01774=1232.816,82.579,-46.181,-178.572,5.437,148.517
C01775=1232.821,82.330,-46.163,-178.574,5.436,148.518
C01776=1232.826,82.061,-46.144,-178.577,5.435,148.519
C01777=1232.831,81.793,-46.125,-178.580,5.435,148.519
C01778=1232.836,81.525,-46.106,-178.582,5.434,148.520
C01779=1232.842,81.256,-46.086,-178.585,5.434,148.521
C01780=1232.847,81.006,-46.067,-178.588,5.433,148.521
C01781=1232.852,80.757,-46.049,-178.590,5.432,148.522
C01782=1232.856,80.508,-46.031,-178.592,5.431,148.522
C01783=1232.861,80.259,-46.013,-178.596,5.430,148.523
C01784=1232.866,80.010,-45.996,-178.598,5.429,148.524
C01785=1232.870,79.761,-45.978,-178.601,5.429,148.524
C01786=1232.876,79.511,-45.961,-178.603,5.428,148.525
C01787=1232.881,79.262,-45.943,-178.606,5.427,148.526
C01788=1232.885,79.013,-45.925,-178.608,5.427,148.526
C01789=1232.890,78.763,-45.906,-178.611,5.426,148.527
C01790=1232.895,78.514,-45.888,-178.613,5.426,148.528
C01791=1232.900,78.265,-45.870,-178.616,5.425,148.528
C01792=1232.905,78.015,-45.852,-178.618,5.424,148.529
C01793=1232.910,77.766,-45.835,-178.621,5.423,148.529
C01794=1232.915,77.516,-45.817,-178.623,5.423,148.530
C01795=1232.920,77.267,-45.799,-178.626,5.422,148.531
C01796=1232.924,77.018,-45.781,-178.629,5.422,148.531
C01797=1232.929,76.769,-45.763,-178.631,5.421,148.532
C01798=1232.935,76.519,-45.746,-178.633,5.420,148.532
C01799=1232.939,76.270,-45.729,-178.636,5.419,148.533
C01800=1232.944,76.021,-45.711,-178.639,5.419,148.534
C01801=1232.949,75.772,-45.693,-178.641,5.418,148.534
C01802=1232.954,75.522,-45.675,-178.643,5.417,148.535
C01803=1232.959,75.273,-45.657,-178.646,5.417,148.535
C01804=1232.964,75.024,-45.639,-178.649,5.416,148.536
C01805=1232.968,74.774,-45.621,-178.651,5.416,148.537
C01806=1232.973,74.524,-45.604,-178.654,5.415,148.537
C01807=1232.977,74.275,-45.586,-178.657,5.414,148.538
C01808=1232.982,74.026,-45.569,-178.659,5.413,148.538
C01809=1232.987,73.776,-45.551,-178.661,5.413,148.539
C01810=1232.992,73.527,-45.533,-178.664,5.412,148.540
C01811=1232.997,73.278,-45.515,-178.667,5.412,148.540
